LIN {X 0,Y 154.212,Z 695.372,A -85,B 0,C 180,E1 -23468.618,E2 -23468.618} C_VEL
LIN {X 0,Y 158.91,Z 697.062,A -85,B 0,C 180,E1 -23463.751,E2 -23463.751} C_VEL
LIN {X 0,Y 164.977,Z 697.541,A -85,B 0,C 180,E1 -23459.256,E2 -23459.256} C_VEL
LIN {X 0,Y 172.53,Z 696.813,A -85,B 0,C 180,E1 -23455.229,E2 -23455.229} C_VEL
LIN {X 0,Y 181.226,Z 694.851,A -85,B 0,C 180,E1 -23451.648,E2 -23451.648} C_VEL
LIN {X 0,Y 190.909,Z 691.562,A -85,B 0,C 180,E1 -23448.498,E2 -23448.498} C_VEL
LIN {X 0,Y 201.458,Z 686.897,A -85,B 0,C 180,E1 -23445.756,E2 -23445.756} C_VEL
LIN {X 0,Y 207.006,Z 684.055,A -85,B 0,C 180,E1 -23444.523,E2 -23444.523} C_VEL
LIN {X 0,Y 204.306,Z 685.314,A -85,B 0,C 180,E1 -23443.471,E2 -23443.471} C_VEL
LIN {X 0,Y 193.798,Z 689.658,A -85,B 0,C 180,E1 -23440.75,E2 -23440.75} C_VEL
LIN {X 0,Y 188.167,Z 691.451,A -85,B 0,C 180,E1 -23439.054,E2 -23439.054} C_VEL
LIN {X 0,Y 183.778,Z 692.639,A -85,B 0,C 180,E1 -23437.875,E2 -23437.875} C_VEL
LIN {X 0,Y 175.524,Z 694.141,A -85,B 0,C 180,E1 -23436.18,E2 -23436.18} C_VEL
LIN {X 0,Y 169.039,Z 694.749,A -85,B 0,C 180,E1 -23434.699,E2 -23434.699} C_VEL
LIN {X 0,Y 164.24,Z 694.773,A -85,B 0,C 180,E1 -23433.024,E2 -23433.024} C_VEL
LIN {X 0,Y 163.677,Z 694.7,A -85,B 0,C 180,E1 -23432.745,E2 -23432.745} C_VEL
LIN {X 0,Y 157.81,Z 693.959,A -85,B 0,C 180,E1 -23429.333,E2 -23429.333} C_VEL
LIN {X 0,Y 151.671,Z 691.836,A -85,B 0,C 180,E1 -23424.648,E2 -23424.648} C_VEL
LIN {X 0,Y 147.172,Z 688.478,A -85,B 0,C 180,E1 -23419.528,E2 -23419.528} C_VEL
LIN {X 0,Y 144.142,Z 683.771,A -85,B 0,C 180,E1 -23414.11,E2 -23414.11} C_VEL
LIN {X 0,Y 142.894,Z 679.29,A -85,B 0,C 180,E1 -23409.92,E2 -23409.92} C_VEL
LIN {X 0,Y 142.444,Z 672.774,A -85,B 0,C 180,E1 -23404.953,E2 -23404.953} C_VEL
LIN {X 0,Y 142.536,Z 665.887,A -85,B 0,C 180,E1 -23400.706,E2 -23400.706} C_VEL
LIN {X 0,Y 142.741,Z 657.173,A -85,B 0,C 180,E1 -23396.471,E2 -23396.471} C_VEL
LIN {X 0,Y 143.135,Z 648.344,A -85,B 0,C 180,E1 -23392.949,E2 -23392.949} C_VEL
LIN {X 0,Y 143.785,Z 637.536,A -85,B 0,C 180,E1 -23389.412,E2 -23389.412} C_VEL
LIN {X 0,Y 144.647,Z 625.917,A -85,B 0,C 180,E1 -23386.348,E2 -23386.348} C_VEL
LIN {X 0,Y 145.649,Z 612.215,A -85,B 0,C 180,E1 -23383.531,E2 -23383.531} C_VEL
LIN {X 0,Y 146.651,Z 597.973,A -85,B 0,C 180,E1 -23381.307,E2 -23381.307} C_VEL
LIN {X 0,Y 147.514,Z 581.99,A -85,B 0,C 180,E1 -23379.52,E2 -23379.52} C_VEL
LIN {X 0,Y 150.866,Z 512.722,A -85,B 0,C 180,E1 -23373.113,E2 -23373.113} C_VEL
LIN {X 0,Y 150.241,Z 506.777,A -85,B 0,C 180,E1 -23372.506,E2 -23372.506} C_VEL
LIN {X 0,Y 150.609,Z 508.356,A -85,B 0,C 180,E1 -23372.079,E2 -23372.079} C_VEL
LIN {X 0,Y 150.906,Z 508.756,A -85,B 0,C 180,E1 -23371.827,E2 -23371.827} C_VEL
LIN {X 0,Y 151.972,Z 508.48,A -85,B 0,C 180,E1 -23371.11,E2 -23371.11} C_VEL
LIN {X 0,Y 153.68,Z 505.488,A -85,B 0,C 180,E1 -23370.25,E2 -23370.25} C_VEL
LIN {X 0,Y 155.859,Z 499.285,A -85,B 0,C 180,E1 -23369.422,E2 -23369.422} C_VEL
LIN {X 0,Y 157.427,Z 493.941,A -85,B 0,C 180,E1 -23368.928,E2 -23368.928} C_VEL
LIN {X 0,Y 159.201,Z 492.39,A -85,B 0,C 180,E1 -23368.011,E2 -23368.011} C_VEL
LIN {X 0,Y 160.868,Z 489.906,A -85,B 0,C 180,E1 -23367.273,E2 -23367.273} C_VEL
LIN {X 0,Y 163.685,Z 491.039,A -85,B 0,C 180,E1 -23365.68,E2 -23365.68} C_VEL
LIN {X 0,Y 168.067,Z 498.093,A -85,B 0,C 180,E1 -23363.05,E2 -23363.05} C_VEL
LIN {X 0,Y 173.181,Z 507.456,A -85,B 0,C 180,E1 -23360.252,E2 -23360.252} C_VEL
LIN {X 0,Y 177.806,Z 517.181,A -85,B 0,C 180,E1 -23357.91,E2 -23357.91} C_VEL
LIN {X 0,Y 181.79,Z 527.34,A -85,B 0,C 180,E1 -23355.965,E2 -23355.965} C_VEL
LIN {X 0,Y 177.677,Z 588.851,A -85,B 0,C 180,E1 -23353.793,E2 -23353.793} C_VEL
LIN {X 0,Y 175.901,Z 602.055,A -85,B 0,C 180,E1 -23353.016,E2 -23353.016} C_VEL
LIN {X 0,Y 173.476,Z 614.981,A -85,B 0,C 180,E1 -23351.754,E2 -23351.754} C_VEL
LIN {X 0,Y 170.268,Z 627.141,A -85,B 0,C 180,E1 -23350.161,E2 -23350.161} C_VEL
LIN {X 0,Y 166.603,Z 638.578,A -85,B 0,C 180,E1 -23348.094,E2 -23348.094} C_VEL
LIN {X 0,Y 162.567,Z 648.859,A -85,B 0,C 180,E1 -23345.706,E2 -23345.706} C_VEL
LIN {X 0,Y 158.622,Z 658.132,A -85,B 0,C 180,E1 -23342.872,E2 -23342.872} C_VEL
LIN {X 0,Y 154.329,Z 667.038,A -85,B 0,C 180,E1 -23339.311,E2 -23339.311} C_VEL
LIN {X 0,Y 150.538,Z 674.209,A -85,B 0,C 180,E1 -23335.585,E2 -23335.585} C_VEL
LIN {X 0,Y 147.715,Z 679.062,A -85,B 0,C 180,E1 -23332.373,E2 -23332.373} C_VEL
LIN {X 0,Y 145.104,Z 683.747,A -85,B 0,C 180,E1 -23328.35,E2 -23328.35} C_VEL
LIN {X 0,Y 143.11,Z 687.318,A -85,B 0,C 180,E1 -23324.214,E2 -23324.214} C_VEL
LIN {X 0,Y 142.13,Z 689.155,A -85,B 0,C 180,E1 -23321.408,E2 -23321.408} C_VEL
LIN {X 0,Y 141.433,Z 690.53,A -85,B 0,C 180,E1 -23318.573,E2 -23318.573} C_VEL
LIN {X 0,Y 140.948,Z 691.502,A -85,B 0,C 180,E1 -23315.723,E2 -23315.723} C_VEL
LIN {X 0,Y 140.653,Z 692.19,A -85,B 0,C 180,E1 -23312.077,E2 -23312.077} C_VEL
LIN {X 0,Y 140.678,Z 692.063,A -85,B 0,C 180,E1 -23307.136,E2 -23307.136} C_VEL
LIN {X 0,Y 140.948,Z 691.453,A -85,B 0,C 180,E1 -23304.277,E2 -23304.277} C_VEL
LIN {X 0,Y 141.434,Z 690.461,A -85,B 0,C 180,E1 -23301.427,E2 -23301.427} C_VEL
LIN {X 0,Y 142.136,Z 689.046,A -85,B 0,C 180,E1 -23298.593,E2 -23298.593} C_VEL
LIN {X 0,Y 143.725,Z 686.118,A -85,B 0,C 180,E1 -23294.398,E2 -23294.398} C_VEL
LIN {X 0,Y 145.972,Z 682.14,A -85,B 0,C 180,E1 -23290.304,E2 -23290.304} C_VEL
LIN {X 0,Y 148.823,Z 676.997,A -85,B 0,C 180,E1 -23286.334,E2 -23286.334} C_VEL
LIN {X 0,Y 152.409,Z 670.519,A -85,B 0,C 180,E1 -23282.54,E2 -23282.54} C_VEL
LIN {X 0,Y 156.116,Z 663.211,A -85,B 0,C 180,E1 -23279.208,E2 -23279.208} C_VEL
LIN {X 0,Y 160.252,Z 654.194,A -85,B 0,C 180,E1 -23276.002,E2 -23276.002} C_VEL
LIN {X 0,Y 164.398,Z 643.98,A -85,B 0,C 180,E1 -23273.237,E2 -23273.237} C_VEL
LIN {X 0,Y 168.474,Z 632.507,A -85,B 0,C 180,E1 -23270.88,E2 -23270.88} C_VEL
LIN {X 0,Y 171.801,Z 621.001,A -85,B 0,C 180,E1 -23269.116,E2 -23269.116} C_VEL
LIN {X 0,Y 174.716,Z 607.936,A -85,B 0,C 180,E1 -23267.641,E2 -23267.641} C_VEL
LIN {X 0,Y 176.804,Z 595.313,A -85,B 0,C 180,E1 -23266.698,E2 -23266.698} C_VEL
LIN {X 0,Y 178.214,Z 580.651,A -85,B 0,C 180,E1 -23266.047,E2 -23266.047} C_VEL
LIN {X 0,Y 181.605,Z 527.022,A -85,B 0,C 180,E1 -23264.154,E2 -23264.154} C_VEL
LIN {X 0,Y 176.964,Z 515.425,A -85,B 0,C 180,E1 -23261.89,E2 -23261.89} C_VEL
LIN {X 0,Y 171.539,Z 504.437,A -85,B 0,C 180,E1 -23259.109,E2 -23259.109} C_VEL
LIN {X 0,Y 166.539,Z 495.65,A -85,B 0,C 180,E1 -23256.31,E2 -23256.31} C_VEL
LIN {X 0,Y 161.218,Z 487.289,A -85,B 0,C 180,E1 -23252.975,E2 -23252.975} C_VEL
LIN {X 0,Y 157.657,Z 482.205,A -85,B 0,C 180,E1 -23250.469,E2 -23250.469} C_VEL
LIN {X 0,Y 156.455,Z 481.134,A -85,B 0,C 180,E1 -23249.612,E2 -23249.612} C_VEL
LIN {X 0,Y 154.858,Z 481.135,A -85,B 0,C 180,E1 -23248.552,E2 -23248.552} C_VEL
LIN {X 0,Y 151.794,Z 488.731,A -85,B 0,C 180,E1 -23247.125,E2 -23247.125} C_VEL
LIN {X 0,Y 150.556,Z 490.586,A -85,B 0,C 180,E1 -23246.383,E2 -23246.383} C_VEL
LIN {X 0,Y 150.161,Z 490.264,A -85,B 0,C 180,E1 -23246.041,E2 -23246.041} C_VEL
LIN {X 0,Y 149.866,Z 488.044,A -85,B 0,C 180,E1 -23245.567,E2 -23245.567} C_VEL
LIN {X 0,Y 149.888,Z 487.183,A -85,B 0,C 180,E1 -23245.49,E2 -23245.49} C_VEL
LIN {X 0,Y 147.247,Z 543.271,A -85,B 0,C 180,E1 -23240.245,E2 -23240.245} C_VEL
LIN {X 0,Y 146.476,Z 557.446,A -85,B 0,C 180,E1 -23238.534,E2 -23238.534} C_VEL
LIN {X 0,Y 145.519,Z 570.062,A -85,B 0,C 180,E1 -23236.484,E2 -23236.484} C_VEL
LIN {X 0,Y 144.607,Z 581.945,A -85,B 0,C 180,E1 -23234.064,E2 -23234.064} C_VEL
LIN {X 0,Y 143.715,Z 594.089,A -85,B 0,C 180,E1 -23230.952,E2 -23230.952} C_VEL
LIN {X 0,Y 142.872,Z 606.339,A -85,B 0,C 180,E1 -23227.064,E2 -23227.064} C_VEL
LIN {X 0,Y 142.527,Z 617.048,A -85,B 0,C 180,E1 -23222.827,E2 -23222.827} C_VEL
LIN {X 0,Y 142.25,Z 625.752,A -85,B 0,C 180,E1 -23218.585,E2 -23218.585} C_VEL
LIN {X 0,Y 142.882,Z 634.154,A -85,B 0,C 180,E1 -23213.646,E2 -23213.646} C_VEL
LIN {X 0,Y 144.638,Z 641.011,A -85,B 0,C 180,E1 -23208.793,E2 -23208.793} C_VEL
LIN {X 0,Y 147.832,Z 647.241,A -85,B 0,C 180,E1 -23203.427,E2 -23203.427} C_VEL
LIN {X 0,Y 152.456,Z 651.936,A -85,B 0,C 180,E1 -23198.359,E2 -23198.359} C_VEL
LIN {X 0,Y 158.523,Z 655.239,A -85,B 0,C 180,E1 -23193.683,E2 -23193.683} C_VEL
LIN {X 0,Y 165.9,Z 657.207,A -85,B 0,C 180,E1 -23189.446,E2 -23189.446} C_VEL
LIN {X 0,Y 174.366,Z 657.834,A -85,B 0,C 180,E1 -23185.647,E2 -23185.647} C_VEL
LIN {X 0,Y 183.656,Z 657.118,A -85,B 0,C 180,E1 -23182.246,E2 -23182.246} C_VEL
LIN {X 0,Y 193.761,Z 655.054,A -85,B 0,C 180,E1 -23179.24,E2 -23179.24} C_VEL
LIN {X 0,Y 198.138,Z 653.804,A -85,B 0,C 180,E1 -23178.094,E2 -23178.094} C_VEL
LIN {X 0,Y 197.395,Z 654.328,A -85,B 0,C 180,E1 -23177.526,E2 -23177.526} C_VEL
LIN {X 0,Y 187.896,Z 658.559,A -85,B 0,C 180,E1 -23175.29,E2 -23175.29} C_VEL
LIN {X 0,Y 177.607,Z 662.342,A -85,B 0,C 180,E1 -23172.276,E2 -23172.276} C_VEL
LIN {X 0,Y 168.371,Z 664.962,A -85,B 0,C 180,E1 -23168.764,E2 -23168.764} C_VEL
LIN {X 0,Y 160.36,Z 666.488,A -85,B 0,C 180,E1 -23164.733,E2 -23164.733} C_VEL
LIN {X 0,Y 156.579,Z 666.915,A -85,B 0,C 180,E1 -23162.304,E2 -23162.304} C_VEL
LIN {X 0,Y 152.872,Z 673.912,A -85,B 0,C 180,E1 -23159.542,E2 -23159.542} C_VEL
LIN {X 0,Y 149.306,Z 681.107,A -85,B 0,C 180,E1 -23155.811,E2 -23155.811} C_VEL
LIN {X 0,Y 146.611,Z 686.073,A -85,B 0,C 180,E1 -23152.55,E2 -23152.55} C_VEL
LIN {X 0,Y 143.991,Z 690.879,A -85,B 0,C 180,E1 -23148.497,E2 -23148.497} C_VEL
LIN {X 0,Y 142.231,Z 694.562,A -85,B 0,C 180,E1 -23144.304,E2 -23144.304} C_VEL
LIN {X 0,Y 141.421,Z 696.462,A -85,B 0,C 180,E1 -23141.466,E2 -23141.466} C_VEL
LIN {X 0,Y 140.866,Z 697.905,A -85,B 0,C 180,E1 -23138.608,E2 -23138.608} C_VEL
LIN {X 0,Y 140.62,Z 698.923,A -85,B 0,C 180,E1 -23135.737,E2 -23135.737} C_VEL
LIN {X 0,Y 140.587,Z 699.723,A -85,B 0,C 180,E1 -23131.109,E2 -23131.109} C_VEL
LIN {X 0,Y 140.592,Z 699.566,A -85,B 0,C 180,E1 -23127.135,E2 -23127.135} C_VEL
LIN {X 0,Y 140.723,Z 698.951,A -85,B 0,C 180,E1 -23124.267,E2 -23124.267} C_VEL
LIN {X 0,Y 141.103,Z 697.946,A -85,B 0,C 180,E1 -23121.406,E2 -23121.406} C_VEL
LIN {X 0,Y 141.854,Z 696.529,A -85,B 0,C 180,E1 -23118.57,E2 -23118.57} C_VEL
LIN {X 0,Y 143.608,Z 693.574,A -85,B 0,C 180,E1 -23114.385,E2 -23114.385} C_VEL
LIN {X 0,Y 145.115,Z 691.541,A -85,B 0,C 180,E1 -23112.016,E2 -23112.016} C_VEL
LIN {X 0,Y 147.719,Z 694.131,A -85,B 0,C 180,E1 -23107.628,E2 -23107.628} C_VEL
LIN {X 0,Y 152.627,Z 696.23,A -85,B 0,C 180,E1 -23102.582,E2 -23102.582} C_VEL
LIN {X 0,Y 158.935,Z 697.158,A -85,B 0,C 180,E1 -23097.952,E2 -23097.952} C_VEL
LIN {X 0,Y 166.768,Z 696.928,A -85,B 0,C 180,E1 -23093.843,E2 -23093.843} C_VEL
LIN {X 0,Y 175.729,Z 695.482,A -85,B 0,C 180,E1 -23090.216,E2 -23090.216} C_VEL
LIN {X 0,Y 185.696,Z 692.789,A -85,B 0,C 180,E1 -23087.059,E2 -23087.059} C_VEL
LIN {X 0,Y 196.536,Z 688.785,A -85,B 0,C 180,E1 -23084.341,E2 -23084.341} C_VEL
LIN {X 0,Y 193.456,Z 689.867,A -85,B 0,C 180,E1 -23083.4,E2 -23083.4} C_VEL
LIN {X 0,Y 183.305,Z 692.742,A -85,B 0,C 180,E1 -23080.598,E2 -23080.598} C_VEL
LIN {X 0,Y 173.834,Z 694.39,A -85,B 0,C 180,E1 -23077.332,E2 -23077.332} C_VEL
LIN {X 0,Y 165.266,Z 694.806,A -85,B 0,C 180,E1 -23073.561,E2 -23073.561} C_VEL
LIN {X 0,Y 163.677,Z 694.7,A -85,B 0,C 180,E1 -23072.745,E2 -23072.745} C_VEL
LIN {X 0,Y 159.962,Z 694.417,A -85,B 0,C 180,E1 -23071.125,E2 -23071.125} C_VEL
LIN {X 0,Y 152.808,Z 693.264,A -85,B 0,C 180,E1 -23068.653,E2 -23068.653} C_VEL
LIN {X 0,Y 146.216,Z 691.291,A -85,B 0,C 180,E1 -23065.935,E2 -23065.935} C_VEL
LIN {X 0,Y 143.474,Z 689.811,A -85,B 0,C 180,E1 -23063.952,E2 -23063.952} C_VEL
LIN {X 0,Y 139.661,Z 686.102,A -85,B 0,C 180,E1 -23059.092,E2 -23059.092} C_VEL
LIN {X 0,Y 137.477,Z 682.117,A -85,B 0,C 180,E1 -23054.809,E2 -23054.809} C_VEL
LIN {X 0,Y 135.917,Z 675.447,A -85,B 0,C 180,E1 -23048.924,E2 -23048.924} C_VEL
LIN {X 0,Y 135.773,Z 669.278,A -85,B 0,C 180,E1 -23044.453,E2 -23044.453} C_VEL
LIN {X 0,Y 135.872,Z 661.615,A -85,B 0,C 180,E1 -23040,E2 -23040} C_VEL
LIN {X 0,Y 136.019,Z 653.838,A -85,B 0,C 180,E1 -23036.297,E2 -23036.297} C_VEL
LIN {X 0,Y 136.443,Z 644.348,A -85,B 0,C 180,E1 -23032.601,E2 -23032.601} C_VEL
LIN {X 0,Y 137.064,Z 634.008,A -85,B 0,C 180,E1 -23029.288,E2 -23029.288} C_VEL
LIN {X 0,Y 137.99,Z 621.727,A -85,B 0,C 180,E1 -23026.098,E2 -23026.098} C_VEL
LIN {X 0,Y 138.833,Z 608.741,A -85,B 0,C 180,E1 -23023.457,E2 -23023.457} C_VEL
LIN {X 0,Y 139.697,Z 596.213,A -85,B 0,C 180,E1 -23021.483,E2 -23021.483} C_VEL
LIN {X 0,Y 140.791,Z 574.293,A -85,B 0,C 180,E1 -23019.07,E2 -23019.07} C_VEL
LIN {X 0,Y 142.444,Z 537.427,A -85,B 0,C 180,E1 -23015.399,E2 -23015.399} C_VEL
LIN {X 0,Y 142.467,Z 540.512,A -85,B 0,C 180,E1 -23015.014,E2 -23015.014} C_VEL
LIN {X 0,Y 142.752,Z 541.298,A -85,B 0,C 180,E1 -23014.678,E2 -23014.678} C_VEL
LIN {X 0,Y 143.433,Z 541.139,A -85,B 0,C 180,E1 -23014.126,E2 -23014.126} C_VEL
LIN {X 0,Y 144.619,Z 538.864,A -85,B 0,C 180,E1 -23013.418,E2 -23013.418} C_VEL
LIN {X 0,Y 146.697,Z 533.23,A -85,B 0,C 180,E1 -23012.416,E2 -23012.416} C_VEL
LIN {X 0,Y 150.453,Z 520.331,A -85,B 0,C 180,E1 -23011.011,E2 -23011.011} C_VEL
LIN {X 0,Y 151.829,Z 515.486,A -85,B 0,C 180,E1 -23010.54,E2 -23010.54} C_VEL
LIN {X 0,Y 153.658,Z 513.922,A -85,B 0,C 180,E1 -23009.493,E2 -23009.493} C_VEL
LIN {X 0,Y 155.826,Z 510.331,A -85,B 0,C 180,E1 -23008.472,E2 -23008.472} C_VEL
LIN {X 0,Y 158.257,Z 504.284,A -85,B 0,C 180,E1 -23007.562,E2 -23007.562} C_VEL
LIN {X 0,Y 159.969,Z 499.081,A -85,B 0,C 180,E1 -23007.026,E2 -23007.026} C_VEL
LIN {X 0,Y 160.998,Z 497.94,A -85,B 0,C 180,E1 -23006.556,E2 -23006.556} C_VEL
LIN {X 0,Y 161.78,Z 498.314,A -85,B 0,C 180,E1 -23006.109,E2 -23006.109} C_VEL
LIN {X 0,Y 166.905,Z 507.229,A -85,B 0,C 180,E1 -23002.939,E2 -23002.939} C_VEL
LIN {X 0,Y 172.163,Z 517.954,A -85,B 0,C 180,E1 -22999.988,E2 -22999.988} C_VEL
LIN {X 0,Y 176.511,Z 528.678,A -85,B 0,C 180,E1 -22997.691,E2 -22997.691} C_VEL
LIN {X 0,Y 176.81,Z 529.477,A -85,B 0,C 180,E1 -22997.537,E2 -22997.537} C_VEL
LIN {X 0,Y 172.614,Z 589.011,A -85,B 0,C 180,E1 -22995.422,E2 -22995.422} C_VEL
LIN {X 0,Y 170.772,Z 602.284,A -85,B 0,C 180,E1 -22994.631,E2 -22994.631} C_VEL
LIN {X 0,Y 168.257,Z 615.138,A -85,B 0,C 180,E1 -22993.361,E2 -22993.361} C_VEL
LIN {X 0,Y 164.903,Z 627.308,A -85,B 0,C 180,E1 -22991.753,E2 -22991.753} C_VEL
LIN {X 0,Y 161.082,Z 638.752,A -85,B 0,C 180,E1 -22989.65,E2 -22989.65} C_VEL
LIN {X 0,Y 156.865,Z 649.036,A -85,B 0,C 180,E1 -22987.217,E2 -22987.217} C_VEL
LIN {X 0,Y 152.7,Z 658.313,A -85,B 0,C 180,E1 -22984.32,E2 -22984.32} C_VEL
LIN {X 0,Y 148.16,Z 667.222,A -85,B 0,C 180,E1 -22980.659,E2 -22980.659} C_VEL
LIN {X 0,Y 144.171,Z 674.394,A -85,B 0,C 180,E1 -22976.803,E2 -22976.803} C_VEL
LIN {X 0,Y 141.161,Z 679.248,A -85,B 0,C 180,E1 -22973.472,E2 -22973.472} C_VEL
LIN {X 0,Y 138.366,Z 683.935,A -85,B 0,C 180,E1 -22969.278,E2 -22969.278} C_VEL
LIN {X 0,Y 136.218,Z 687.506,A -85,B 0,C 180,E1 -22964.95,E2 -22964.95} C_VEL
LIN {X 0,Y 135.166,Z 689.343,A -85,B 0,C 180,E1 -22962.004,E2 -22962.004} C_VEL
LIN {X 0,Y 134.426,Z 690.718,A -85,B 0,C 180,E1 -22959.024,E2 -22959.024} C_VEL
LIN {X 0,Y 133.603,Z 692.281,A -85,B 0,C 180,E1 -22953.015,E2 -22953.015} C_VEL
LIN {X 0,Y 133.542,Z 692.447,A -85,B 0,C 180,E1 -22949.322,E2 -22949.322} C_VEL
LIN {X 0,Y 133.882,Z 691.642,A -85,B 0,C 180,E1 -22943.974,E2 -22943.974} C_VEL
LIN {X 0,Y 134.427,Z 690.65,A -85,B 0,C 180,E1 -22940.976,E2 -22940.976} C_VEL
LIN {X 0,Y 135.171,Z 689.236,A -85,B 0,C 180,E1 -22937.996,E2 -22937.996} C_VEL
LIN {X 0,Y 136.881,Z 686.308,A -85,B 0,C 180,E1 -22933.597,E2 -22933.597} C_VEL
LIN {X 0,Y 139.3,Z 682.329,A -85,B 0,C 180,E1 -22929.319,E2 -22929.319} C_VEL
LIN {X 0,Y 142.337,Z 677.186,A -85,B 0,C 180,E1 -22925.185,E2 -22925.185} C_VEL
LIN {X 0,Y 146.138,Z 670.707,A -85,B 0,C 180,E1 -22921.255,E2 -22921.255} C_VEL
LIN {X 0,Y 149.799,Z 663.881,A -85,B 0,C 180,E1 -22918.02,E2 -22918.02} C_VEL
LIN {X 0,Y 154.401,Z 654.38,A -85,B 0,C 180,E1 -22914.524,E2 -22914.524} C_VEL
LIN {X 0,Y 158.767,Z 644.164,A -85,B 0,C 180,E1 -22911.704,E2 -22911.704} C_VEL
LIN {X 0,Y 163.031,Z 632.687,A -85,B 0,C 180,E1 -22909.306,E2 -22909.306} C_VEL
LIN {X 0,Y 166.503,Z 621.176,A -85,B 0,C 180,E1 -22907.518,E2 -22907.518} C_VEL
LIN {X 0,Y 169.554,Z 608.102,A -85,B 0,C 180,E1 -22906.029,E2 -22906.029} C_VEL
LIN {X 0,Y 171.754,Z 595.181,A -85,B 0,C 180,E1 -22905.061,E2 -22905.061} C_VEL
LIN {X 0,Y 173.126,Z 581.338,A -85,B 0,C 180,E1 -22904.434,E2 -22904.434} C_VEL
LIN {X 0,Y 176.594,Z 529.191,A -85,B 0,C 180,E1 -22902.576,E2 -22902.576} C_VEL
LIN {X 0,Y 172.028,Z 517.825,A -85,B 0,C 180,E1 -22900.17,E2 -22900.17} C_VEL
LIN {X 0,Y 166.417,Z 506.429,A -85,B 0,C 180,E1 -22897.019,E2 -22897.019} C_VEL
LIN {X 0,Y 161.385,Z 497.781,A -85,B 0,C 180,E1 -22893.899,E2 -22893.899} C_VEL
LIN {X 0,Y 158.043,Z 492.469,A -85,B 0,C 180,E1 -22891.594,E2 -22891.594} C_VEL
LIN {X 0,Y 156.017,Z 489.33,A -85,B 0,C 180,E1 -22890.076,E2 -22890.076} C_VEL
LIN {X 0,Y 155.57,Z 489.422,A -85,B 0,C 180,E1 -22889.798,E2 -22889.798} C_VEL
LIN {X 0,Y 153.336,Z 494.268,A -85,B 0,C 180,E1 -22888.768,E2 -22888.768} C_VEL
LIN {X 0,Y 151.403,Z 496.822,A -85,B 0,C 180,E1 -22887.658,E2 -22887.658} C_VEL
LIN {X 0,Y 150.779,Z 497.545,A -85,B 0,C 180,E1 -22887.274,E2 -22887.274} C_VEL
LIN {X 0,Y 146.646,Z 513.67,A -85,B 0,C 180,E1 -22885.786,E2 -22885.786} C_VEL
LIN {X 0,Y 143.957,Z 522.395,A -85,B 0,C 180,E1 -22884.518,E2 -22884.518} C_VEL
LIN {X 0,Y 142.335,Z 526.521,A -85,B 0,C 180,E1 -22883.556,E2 -22883.556} C_VEL
LIN {X 0,Y 141.607,Z 527.608,A -85,B 0,C 180,E1 -22883.007,E2 -22883.007} C_VEL
LIN {X 0,Y 141.19,Z 527.548,A -85,B 0,C 180,E1 -22882.595,E2 -22882.595} C_VEL
LIN {X 0,Y 140.98,Z 526.456,A -85,B 0,C 180,E1 -22882.244,E2 -22882.244} C_VEL
LIN {X 0,Y 140.994,Z 524.168,A -85,B 0,C 180,E1 -22881.953,E2 -22881.953} C_VEL
LIN {X 0,Y 139.847,Z 549.609,A -85,B 0,C 180,E1 -22879.257,E2 -22879.257} C_VEL
LIN {X 0,Y 139.032,Z 563.216,A -85,B 0,C 180,E1 -22877.276,E2 -22877.276} C_VEL
LIN {X 0,Y 137.983,Z 577.082,A -85,B 0,C 180,E1 -22874.591,E2 -22874.591} C_VEL
LIN {X 0,Y 136.961,Z 589.624,A -85,B 0,C 180,E1 -22871.5,E2 -22871.5} C_VEL
LIN {X 0,Y 136.186,Z 601.705,A -85,B 0,C 180,E1 -22867.786,E2 -22867.786} C_VEL
LIN {X 0,Y 135.732,Z 612.478,A -85,B 0,C 180,E1 -22863.711,E2 -22863.711} C_VEL
LIN {X 0,Y 135.483,Z 620.581,A -85,B 0,C 180,E1 -22860,E2 -22860} C_VEL
LIN {X 0,Y 135.748,Z 629.985,A -85,B 0,C 180,E1 -22854.802,E2 -22854.802} C_VEL
LIN {X 0,Y 137.204,Z 637.739,A -85,B 0,C 180,E1 -22849.672,E2 -22849.672} C_VEL
LIN {X 0,Y 140.136,Z 644.818,A -85,B 0,C 180,E1 -22843.988,E2 -22843.988} C_VEL
LIN {X 0,Y 144.567,Z 650.369,A -85,B 0,C 180,E1 -22838.617,E2 -22838.617} C_VEL
LIN {X 0,Y 148.887,Z 653.572,A -85,B 0,C 180,E1 -22834.86,E2 -22834.86} C_VEL
LIN {X 0,Y 155.887,Z 656.699,A -85,B 0,C 180,E1 -22830.269,E2 -22830.269} C_VEL
LIN {X 0,Y 164.104,Z 658.505,A -85,B 0,C 180,E1 -22826.169,E2 -22826.169} C_VEL
LIN {X 0,Y 173.306,Z 658.97,A -85,B 0,C 180,E1 -22822.534,E2 -22822.534} C_VEL
LIN {X 0,Y 183.318,Z 658.145,A -85,B 0,C 180,E1 -22819.327,E2 -22819.327} C_VEL
LIN {X 0,Y 187.224,Z 657.511,A -85,B 0,C 180,E1 -22818.255,E2 -22818.255} C_VEL
LIN {X 0,Y 186.542,Z 657.918,A -85,B 0,C 180,E1 -22817.722,E2 -22817.722} C_VEL
LIN {X 0,Y 177.579,Z 660.923,A -85,B 0,C 180,E1 -22815.429,E2 -22815.429} C_VEL
LIN {X 0,Y 167.545,Z 663.573,A -85,B 0,C 180,E1 -22812.156,E2 -22812.156} C_VEL
LIN {X 0,Y 158.61,Z 665.153,A -85,B 0,C 180,E1 -22808.341,E2 -22808.341} C_VEL
LIN {X 0,Y 151.228,Z 665.722,A -85,B 0,C 180,E1 -22804.096,E2 -22804.096} C_VEL
LIN {X 0,Y 146.796,Z 673.591,A -85,B 0,C 180,E1 -22800.975,E2 -22800.975} C_VEL
LIN {X 0,Y 142.926,Z 680.918,A -85,B 0,C 180,E1 -22797.055,E2 -22797.055} C_VEL
LIN {X 0,Y 140.03,Z 685.882,A -85,B 0,C 180,E1 -22793.673,E2 -22793.673} C_VEL
LIN {X 0,Y 137.249,Z 690.689,A -85,B 0,C 180,E1 -22789.441,E2 -22789.441} C_VEL
LIN {X 0,Y 135.333,Z 694.372,A -85,B 0,C 180,E1 -22785.05,E2 -22785.05} C_VEL
LIN {X 0,Y 134.452,Z 696.272,A -85,B 0,C 180,E1 -22782.069,E2 -22782.069} C_VEL
LIN {X 0,Y 133.838,Z 697.715,A -85,B 0,C 180,E1 -22779.064,E2 -22779.064} C_VEL
LIN {X 0,Y 133.545,Z 698.734,A -85,B 0,C 180,E1 -22776.042,E2 -22776.042} C_VEL
LIN {X 0,Y 133.542,Z 699.562,A -85,B 0,C 180,E1 -22770.678,E2 -22770.678} C_VEL
LIN {X 0,Y 133.516,Z 699.378,A -85,B 0,C 180,E1 -22766.983,E2 -22766.983} C_VEL
LIN {X 0,Y 134.09,Z 697.757,A -85,B 0,C 180,E1 -22760.953,E2 -22760.953} C_VEL
LIN {X 0,Y 134.889,Z 696.34,A -85,B 0,C 180,E1 -22757.971,E2 -22757.971} C_VEL
LIN {X 0,Y 136.782,Z 693.387,A -85,B 0,C 180,E1 -22753.585,E2 -22753.585} C_VEL
LIN {X 0,Y 139.033,Z 690.433,A -85,B 0,C 180,E1 -22750.242,E2 -22750.242} C_VEL
LIN {X 0,Y 141.33,Z 692.675,A -85,B 0,C 180,E1 -22746.558,E2 -22746.558} C_VEL
LIN {X 0,Y 146.414,Z 695.214,A -85,B 0,C 180,E1 -22741.314,E2 -22741.314} C_VEL
LIN {X 0,Y 152.984,Z 696.583,A -85,B 0,C 180,E1 -22736.545,E2 -22736.545} C_VEL
LIN {X 0,Y 161.111,Z 696.837,A -85,B 0,C 180,E1 -22732.359,E2 -22732.359} C_VEL
LIN {X 0,Y 170.339,Z 695.913,A -85,B 0,C 180,E1 -22728.689,E2 -22728.689} C_VEL
LIN {X 0,Y 180.587,Z 693.78,A -85,B 0,C 180,E1 -22725.531,E2 -22725.531} C_VEL
LIN {X 0,Y 184.301,Z 692.801,A -85,B 0,C 180,E1 -22724.569,E2 -22724.569} C_VEL
LIN {X 0,Y 184.562,Z 692.659,A -85,B 0,C 180,E1 -22723.876,E2 -22723.876} C_VEL
LIN {X 0,Y 178.164,Z 693.928,A -85,B 0,C 180,E1 -22722.113,E2 -22722.113} C_VEL
LIN {X 0,Y 168.263,Z 695.055,A -85,B 0,C 180,E1 -22718.794,E2 -22718.794} C_VEL
LIN {X 0,Y 159.421,Z 694.938,A -85,B 0,C 180,E1 -22714.967,E2 -22714.967} C_VEL
LIN {X 0,Y 151.678,Z 693.613,A -85,B 0,C 180,E1 -22710.643,E2 -22710.643} C_VEL
LIN {X 0,Y 145.303,Z 691.046,A -85,B 0,C 180,E1 -22705.805,E2 -22705.805} C_VEL
LIN {X 0,Y 143.474,Z 689.811,A -85,B 0,C 180,E1 -22703.952,E2 -22703.952} C_VEL
LIN {X 0,Y 141.015,Z 688.176,A -85,B 0,C 180,E1 -22701.897,E2 -22701.897} C_VEL
LIN {X 0,Y 133.941,Z 682.936,A -85,B 0,C 180,E1 -22697.419,E2 -22697.419} C_VEL
LIN {X 0,Y 130.858,Z 679.413,A -85,B 0,C 180,E1 -22694.646,E2 -22694.646} C_VEL
LIN {X 0,Y 130.089,Z 677.629,A -85,B 0,C 180,E1 -22693.13,E2 -22693.13} C_VEL
LIN {X 0,Y 129.138,Z 670.013,A -85,B 0,C 180,E1 -22687.033,E2 -22687.033} C_VEL
LIN {X 0,Y 129.161,Z 664.108,A -85,B 0,C 180,E1 -22683.119,E2 -22683.119} C_VEL
LIN {X 0,Y 129.246,Z 656.887,A -85,B 0,C 180,E1 -22679.221,E2 -22679.221} C_VEL
LIN {X 0,Y 129.474,Z 648.234,A -85,B 0,C 180,E1 -22675.33,E2 -22675.33} C_VEL
LIN {X 0,Y 130.037,Z 636.539,A -85,B 0,C 180,E1 -22671.061,E2 -22671.061} C_VEL
LIN {X 0,Y 130.716,Z 625.962,A -85,B 0,C 180,E1 -22667.975,E2 -22667.975} C_VEL
LIN {X 0,Y 131.496,Z 614.006,A -85,B 0,C 180,E1 -22665.173,E2 -22665.173} C_VEL
LIN {X 0,Y 132.338,Z 601.59,A -85,B 0,C 180,E1 -22662.858,E2 -22662.858} C_VEL
LIN {X 0,Y 133.089,Z 587.635,A -85,B 0,C 180,E1 -22660.929,E2 -22660.929} C_VEL
LIN {X 0,Y 133.823,Z 572.991,A -85,B 0,C 180,E1 -22659.288,E2 -22659.288} C_VEL
LIN {X 0,Y 133.65,Z 576.027,A -85,B 0,C 180,E1 -22659.008,E2 -22659.008} C_VEL
LIN {X 0,Y 133.801,Z 577.477,A -85,B 0,C 180,E1 -22658.629,E2 -22658.629} C_VEL
LIN {X 0,Y 134.263,Z 577.671,A -85,B 0,C 180,E1 -22658.102,E2 -22658.102} C_VEL
LIN {X 0,Y 135.318,Z 575.703,A -85,B 0,C 180,E1 -22657.277,E2 -22657.277} C_VEL
LIN {X 0,Y 137.796,Z 568.432,A -85,B 0,C 180,E1 -22655.819,E2 -22655.819} C_VEL
LIN {X 0,Y 141.164,Z 556.186,A -85,B 0,C 180,E1 -22654.307,E2 -22654.307} C_VEL
LIN {X 0,Y 143.215,Z 548.163,A -85,B 0,C 180,E1 -22653.52,E2 -22653.52} C_VEL
LIN {X 0,Y 144.752,Z 546.737,A -85,B 0,C 180,E1 -22652.471,E2 -22652.471} C_VEL
LIN {X 0,Y 146.703,Z 543.371,A -85,B 0,C 180,E1 -22651.376,E2 -22651.376} C_VEL
LIN {X 0,Y 149.213,Z 536.921,A -85,B 0,C 180,E1 -22650.262,E2 -22650.262} C_VEL
LIN {X 0,Y 152.764,Z 525.481,A -85,B 0,C 180,E1 -22649.014,E2 -22649.014} C_VEL
LIN {X 0,Y 154.101,Z 520.807,A -85,B 0,C 180,E1 -22648.603,E2 -22648.603} C_VEL
LIN {X 0,Y 156.564,Z 517.76,A -85,B 0,C 180,E1 -22647.407,E2 -22647.407} C_VEL
LIN {X 0,Y 159.063,Z 513.27,A -85,B 0,C 180,E1 -22646.38,E2 -22646.38} C_VEL
LIN {X 0,Y 161.18,Z 508.139,A -85,B 0,C 180,E1 -22645.658,E2 -22645.658} C_VEL
LIN {X 0,Y 165.425,Z 516.305,A -85,B 0,C 180,E1 -22642.976,E2 -22642.976} C_VEL
LIN {X 0,Y 169.869,Z 526.241,A -85,B 0,C 180,E1 -22640.378,E2 -22640.378} C_VEL
LIN {X 0,Y 171.942,Z 531.703,A -85,B 0,C 180,E1 -22639.205,E2 -22639.205} C_VEL
LIN {X 0,Y 167.689,Z 589.34,A -85,B 0,C 180,E1 -22637.137,E2 -22637.137} C_VEL
LIN {X 0,Y 165.789,Z 602.519,A -85,B 0,C 180,E1 -22636.343,E2 -22636.343} C_VEL
LIN {X 0,Y 163.175,Z 615.294,A -85,B 0,C 180,E1 -22635.07,E2 -22635.07} C_VEL
LIN {X 0,Y 159.678,Z 627.475,A -85,B 0,C 180,E1 -22633.449,E2 -22633.449} C_VEL
LIN {X 0,Y 155.691,Z 638.925,A -85,B 0,C 180,E1 -22631.314,E2 -22631.314} C_VEL
LIN {X 0,Y 151.273,Z 649.214,A -85,B 0,C 180,E1 -22628.844,E2 -22628.844} C_VEL
LIN {X 0,Y 146.872,Z 658.495,A -85,B 0,C 180,E1 -22625.886,E2 -22625.886} C_VEL
LIN {X 0,Y 142.08,Z 667.406,A -85,B 0,C 180,E1 -22622.124,E2 -22622.124} C_VEL
LIN {X 0,Y 137.87,Z 674.578,A -85,B 0,C 180,E1 -22618.133,E2 -22618.133} C_VEL
LIN {X 0,Y 134.669,Z 679.435,A -85,B 0,C 180,E1 -22614.677,E2 -22614.677} C_VEL
LIN {X 0,Y 131.677,Z 684.122,A -85,B 0,C 180,E1 -22610.299,E2 -22610.299} C_VEL
LIN {X 0,Y 129.361,Z 687.694,A -85,B 0,C 180,E1 -22605.762,E2 -22605.762} C_VEL
LIN {X 0,Y 128.229,Z 689.531,A -85,B 0,C 180,E1 -22602.664,E2 -22602.664} C_VEL
LIN {X 0,Y 127.413,Z 690.907,A -85,B 0,C 180,E1 -22599.525,E2 -22599.525} C_VEL
LIN {X 0,Y 126.515,Z 692.47,A -85,B 0,C 180,E1 -22593.184,E2 -22593.184} C_VEL
LIN {X 0,Y 126.474,Z 692.668,A -85,B 0,C 180,E1 -22590,E2 -22590} C_VEL
LIN {X 0,Y 126.83,Z 691.831,A -85,B 0,C 180,E1 -22583.637,E2 -22583.637} C_VEL
LIN {X 0,Y 127.414,Z 690.839,A -85,B 0,C 180,E1 -22580.475,E2 -22580.475} C_VEL
LIN {X 0,Y 128.234,Z 689.426,A -85,B 0,C 180,E1 -22577.337,E2 -22577.337} C_VEL
LIN {X 0,Y 130.068,Z 686.498,A -85,B 0,C 180,E1 -22572.711,E2 -22572.711} C_VEL
LIN {X 0,Y 132.678,Z 682.519,A -85,B 0,C 180,E1 -22568.235,E2 -22568.235} C_VEL
LIN {X 0,Y 135.92,Z 677.375,A -85,B 0,C 180,E1 -22563.927,E2 -22563.927} C_VEL
LIN {X 0,Y 139.95,Z 670.895,A -85,B 0,C 180,E1 -22559.856,E2 -22559.856} C_VEL
LIN {X 0,Y 144.464,Z 662.864,A -85,B 0,C 180,E1 -22555.997,E2 -22555.997} C_VEL
LIN {X 0,Y 148.665,Z 654.566,A -85,B 0,C 180,E1 -22552.933,E2 -22552.933} C_VEL
LIN {X 0,Y 153.272,Z 644.347,A -85,B 0,C 180,E1 -22550.063,E2 -22550.063} C_VEL
LIN {X 0,Y 157.71,Z 632.867,A -85,B 0,C 180,E1 -22547.622,E2 -22547.622} C_VEL
LIN {X 0,Y 161.339,Z 621.351,A -85,B 0,C 180,E1 -22545.815,E2 -22545.815} C_VEL
LIN {X 0,Y 164.536,Z 608.268,A -85,B 0,C 180,E1 -22544.319,E2 -22544.319} C_VEL
LIN {X 0,Y 166.744,Z 595.834,A -85,B 0,C 180,E1 -22543.37,E2 -22543.37} C_VEL
LIN {X 0,Y 168.275,Z 581.054,A -85,B 0,C 180,E1 -22542.7,E2 -22542.7} C_VEL
LIN {X 0,Y 171.715,Z 531.461,A -85,B 0,C 180,E1 -22540.909,E2 -22540.909} C_VEL
LIN {X 0,Y 167.619,Z 521.198,A -85,B 0,C 180,E1 -22538.572,E2 -22538.572} C_VEL
LIN {X 0,Y 162.716,Z 511.025,A -85,B 0,C 180,E1 -22535.592,E2 -22535.592} C_VEL
LIN {X 0,Y 158.232,Z 503.065,A -85,B 0,C 180,E1 -22532.595,E2 -22532.595} C_VEL
LIN {X 0,Y 155.776,Z 498.924,A -85,B 0,C 180,E1 -22530.783,E2 -22530.783} C_VEL
LIN {X 0,Y 155.462,Z 498.938,A -85,B 0,C 180,E1 -22530.589,E2 -22530.589} C_VEL
LIN {X 0,Y 153.135,Z 502.187,A -85,B 0,C 180,E1 -22529.383,E2 -22529.383} C_VEL
LIN {X 0,Y 148.907,Z 517.733,A -85,B 0,C 180,E1 -22527.954,E2 -22527.954} C_VEL
LIN {X 0,Y 146.031,Z 526.443,A -85,B 0,C 180,E1 -22526.692,E2 -22526.692} C_VEL
LIN {X 0,Y 143.992,Z 531.235,A -85,B 0,C 180,E1 -22525.572,E2 -22525.572} C_VEL
LIN {X 0,Y 142.324,Z 533.759,A -85,B 0,C 180,E1 -22524.429,E2 -22524.429} C_VEL
LIN {X 0,Y 141.505,Z 534.678,A -85,B 0,C 180,E1 -22523.8,E2 -22523.8} C_VEL
LIN {X 0,Y 138.142,Z 548.506,A -85,B 0,C 180,E1 -22522.332,E2 -22522.332} C_VEL
LIN {X 0,Y 135.547,Z 557.291,A -85,B 0,C 180,E1 -22520.806,E2 -22520.806} C_VEL
LIN {X 0,Y 133.646,Z 562.49,A -85,B 0,C 180,E1 -22519.378,E2 -22519.378} C_VEL
LIN {X 0,Y 132.521,Z 564.816,A -85,B 0,C 180,E1 -22518.334,E2 -22518.334} C_VEL
LIN {X 0,Y 132.035,Z 565.154,A -85,B 0,C 180,E1 -22517.742,E2 -22517.742} C_VEL
LIN {X 0,Y 131.889,Z 564.238,A -85,B 0,C 180,E1 -22517.377,E2 -22517.377} C_VEL
LIN {X 0,Y 132.139,Z 561.209,A -85,B 0,C 180,E1 -22517.124,E2 -22517.124} C_VEL
LIN {X 0,Y 131.078,Z 575.331,A -85,B 0,C 180,E1 -22514.353,E2 -22514.353} C_VEL
LIN {X 0,Y 130.02,Z 588.929,A -85,B 0,C 180,E1 -22510.905,E2 -22510.905} C_VEL
LIN {X 0,Y 129.269,Z 601.029,A -85,B 0,C 180,E1 -22507.027,E2 -22507.027} C_VEL
LIN {X 0,Y 128.933,Z 611.078,A -85,B 0,C 180,E1 -22503.125,E2 -22503.125} C_VEL
LIN {X 0,Y 128.693,Z 619.37,A -85,B 0,C 180,E1 -22499.218,E2 -22499.218} C_VEL
LIN {X 0,Y 129.059,Z 629.053,A -85,B 0,C 180,E1 -22493.748,E2 -22493.748} C_VEL
LIN {X 0,Y 130.7,Z 637.035,A -85,B 0,C 180,E1 -22488.367,E2 -22488.367} C_VEL
LIN {X 0,Y 133.431,Z 643.589,A -85,B 0,C 180,E1 -22483.161,E2 -22483.161} C_VEL
LIN {X 0,Y 138.012,Z 649.62,A -85,B 0,C 180,E1 -22477.547,E2 -22477.547} C_VEL
LIN {X 0,Y 142.51,Z 653.179,A -85,B 0,C 180,E1 -22473.651,E2 -22473.651} C_VEL
LIN {X 0,Y 149.757,Z 656.801,A -85,B 0,C 180,E1 -22468.921,E2 -22468.921} C_VEL
LIN {X 0,Y 158.264,Z 659.096,A -85,B 0,C 180,E1 -22464.74,E2 -22464.74} C_VEL
LIN {X 0,Y 167.779,Z 660.095,A -85,B 0,C 180,E1 -22461.073,E2 -22461.073} C_VEL
LIN {X 0,Y 175.758,Z 660.017,A -85,B 0,C 180,E1 -22458.55,E2 -22458.55} C_VEL
LIN {X 0,Y 174.661,Z 660.542,A -85,B 0,C 180,E1 -22457.631,E2 -22457.631} C_VEL
LIN {X 0,Y 167.388,Z 662.213,A -85,B 0,C 180,E1 -22455.543,E2 -22455.543} C_VEL
LIN {X 0,Y 157.609,Z 663.819,A -85,B 0,C 180,E1 -22451.98,E2 -22451.98} C_VEL
LIN {X 0,Y 149.016,Z 664.423,A -85,B 0,C 180,E1 -22447.815,E2 -22447.815} C_VEL
LIN {X 0,Y 146.053,Z 664.507,A -85,B 0,C 180,E1 -22446.012,E2 -22446.012} C_VEL
LIN {X 0,Y 141.555,Z 672.047,A -85,B 0,C 180,E1 -22443.102,E2 -22443.102} C_VEL
LIN {X 0,Y 137.639,Z 678.888,A -85,B 0,C 180,E1 -22439.568,E2 -22439.568} C_VEL
LIN {X 0,Y 134.673,Z 683.828,A -85,B 0,C 180,E1 -22436.332,E2 -22436.332} C_VEL
LIN {X 0,Y 131.476,Z 689.049,A -85,B 0,C 180,E1 -22431.974,E2 -22431.974} C_VEL
LIN {X 0,Y 129.037,Z 693.093,A -85,B 0,C 180,E1 -22427.431,E2 -22427.431} C_VEL
LIN {X 0,Y 127.479,Z 696.082,A -85,B 0,C 180,E1 -22422.74,E2 -22422.74} C_VEL
LIN {X 0,Y 126.805,Z 697.525,A -85,B 0,C 180,E1 -22419.571,E2 -22419.571} C_VEL
LIN {X 0,Y 126.465,Z 698.544,A -85,B 0,C 180,E1 -22416.381,E2 -22416.381} C_VEL
LIN {X 0,Y 126.378,Z 699.172,A -85,B 0,C 180,E1 -22413.188,E2 -22413.188} C_VEL
LIN {X 0,Y 126.504,Z 699.406,A -85,B 0,C 180,E1 -22410,E2 -22410} C_VEL
LIN {X 0,Y 126.444,Z 699.189,A -85,B 0,C 180,E1 -22406.814,E2 -22406.814} C_VEL
LIN {X 0,Y 127.076,Z 697.569,A -85,B 0,C 180,E1 -22400.449,E2 -22400.449} C_VEL
LIN {X 0,Y 127.951,Z 696.152,A -85,B 0,C 180,E1 -22397.308,E2 -22397.308} C_VEL
LIN {X 0,Y 129.992,Z 693.2,A -85,B 0,C 180,E1 -22392.701,E2 -22392.701} C_VEL
LIN {X 0,Y 133.189,Z 689.225,A -85,B 0,C 180,E1 -22388.221,E2 -22388.221} C_VEL
LIN {X 0,Y 137.494,Z 692.673,A -85,B 0,C 180,E1 -22382.61,E2 -22382.61} C_VEL
LIN {X 0,Y 143.506,Z 695.024,A -85,B 0,C 180,E1 -22377.404,E2 -22377.404} C_VEL
LIN {X 0,Y 151.207,Z 696.297,A -85,B 0,C 180,E1 -22372.826,E2 -22372.826} C_VEL
LIN {X 0,Y 160.2,Z 696.462,A -85,B 0,C 180,E1 -22368.848,E2 -22368.848} C_VEL
LIN {X 0,Y 170.225,Z 695.479,A -85,B 0,C 180,E1 -22365.423,E2 -22365.423} C_VEL
LIN {X 0,Y 173.458,Z 694.963,A -85,B 0,C 180,E1 -22364.504,E2 -22364.504} C_VEL
LIN {X 0,Y 173.004,Z 694.933,A -85,B 0,C 180,E1 -22363.677,E2 -22363.677} C_VEL
LIN {X 0,Y 162.811,Z 695.497,A -85,B 0,C 180,E1 -22360.353,E2 -22360.353} C_VEL
LIN {X 0,Y 153.667,Z 694.864,A -85,B 0,C 180,E1 -22356.481,E2 -22356.481} C_VEL
LIN {X 0,Y 145.653,Z 693.04,A -85,B 0,C 180,E1 -22352.057,E2 -22352.057} C_VEL
LIN {X 0,Y 139.035,Z 690.034,A -85,B 0,C 180,E1 -22347.061,E2 -22347.061} C_VEL
LIN {X 0,Y 134.117,Z 685.815,A -85,B 0,C 180,E1 -22341.519,E2 -22341.519} C_VEL
LIN {X 0,Y 130.886,Z 680.227,A -85,B 0,C 180,E1 -22335.574,E2 -22335.574} C_VEL
LIN {X 0,Y 130.089,Z 677.629,A -85,B 0,C 180,E1 -22333.13,E2 -22333.13} C_VEL
LIN {X 0,Y 128.984,Z 674.776,A -85,B 0,C 180,E1 -22330.905,E2 -22330.905} C_VEL
LIN {X 0,Y 125.956,Z 669.1,A -85,B 0,C 180,E1 -22327.514,E2 -22327.514} C_VEL
LIN {X 0,Y 123.633,Z 664.045,A -85,B 0,C 180,E1 -22324.845,E2 -22324.845} C_VEL
LIN {X 0,Y 122.693,Z 660.141,A -85,B 0,C 180,E1 -22322.769,E2 -22322.769} C_VEL
LIN {X 0,Y 122.634,Z 658.846,A -85,B 0,C 180,E1 -22322.058,E2 -22322.058} C_VEL
LIN {X 0,Y 122.668,Z 651.631,A -85,B 0,C 180,E1 -22318.358,E2 -22318.358} C_VEL
LIN {X 0,Y 122.965,Z 641.879,A -85,B 0,C 180,E1 -22314.259,E2 -22314.259} C_VEL
LIN {X 0,Y 123.466,Z 631.253,A -85,B 0,C 180,E1 -22310.581,E2 -22310.581} C_VEL
LIN {X 0,Y 124.224,Z 619.721,A -85,B 0,C 180,E1 -22307.336,E2 -22307.336} C_VEL
LIN {X 0,Y 124.965,Z 606.952,A -85,B 0,C 180,E1 -22304.511,E2 -22304.511} C_VEL
LIN {X 0,Y 125.243,Z 603.053,A -85,B 0,C 180,E1 -22303.705,E2 -22303.705} C_VEL
LIN {X 0,Y 125.041,Z 604.85,A -85,B 0,C 180,E1 -22303.216,E2 -22303.216} C_VEL
LIN {X 0,Y 125.186,Z 605.308,A -85,B 0,C 180,E1 -22302.773,E2 -22302.773} C_VEL
LIN {X 0,Y 126.015,Z 604.847,A -85,B 0,C 180,E1 -22301.778,E2 -22301.778} C_VEL
LIN {X 0,Y 127.541,Z 602.607,A -85,B 0,C 180,E1 -22300.589,E2 -22300.589} C_VEL
LIN {X 0,Y 129.984,Z 597.52,A -85,B 0,C 180,E1 -22299.217,E2 -22299.217} C_VEL
LIN {X 0,Y 132.442,Z 590.41,A -85,B 0,C 180,E1 -22298.092,E2 -22298.092} C_VEL
LIN {X 0,Y 133.965,Z 584.643,A -85,B 0,C 180,E1 -22297.441,E2 -22297.441} C_VEL
LIN {X 0,Y 135.536,Z 582.999,A -85,B 0,C 180,E1 -22296.102,E2 -22296.102} C_VEL
LIN {X 0,Y 137.316,Z 579.55,A -85,B 0,C 180,E1 -22294.888,E2 -22294.888} C_VEL
LIN {X 0,Y 140.222,Z 571.399,A -85,B 0,C 180,E1 -22293.359,E2 -22293.359} C_VEL
LIN {X 0,Y 143.73,Z 559.289,A -85,B 0,C 180,E1 -22291.925,E2 -22291.925} C_VEL
LIN {X 0,Y 145.307,Z 553.387,A -85,B 0,C 180,E1 -22291.371,E2 -22291.371} C_VEL
LIN {X 0,Y 147.835,Z 549.849,A -85,B 0,C 180,E1 -22289.957,E2 -22289.957} C_VEL
LIN {X 0,Y 150.045,Z 545.36,A -85,B 0,C 180,E1 -22288.931,E2 -22288.931} C_VEL
LIN {X 0,Y 153.022,Z 537.514,A -85,B 0,C 180,E1 -22287.797,E2 -22287.797} C_VEL
LIN {X 0,Y 156.918,Z 525.276,A -85,B 0,C 180,E1 -22286.586,E2 -22286.586} C_VEL
LIN {X 0,Y 160.319,Z 520.362,A -85,B 0,C 180,E1 -22285.159,E2 -22285.159} C_VEL
LIN {X 0,Y 161.063,Z 519.391,A -85,B 0,C 180,E1 -22284.853,E2 -22284.853} C_VEL
LIN {X 0,Y 165.698,Z 529.964,A -85,B 0,C 180,E1 -22281.898,E2 -22281.898} C_VEL
LIN {X 0,Y 167.16,Z 533.953,A -85,B 0,C 180,E1 -22280.994,E2 -22280.994} C_VEL
LIN {X 0,Y 165.772,Z 553.605,A -85,B 0,C 180,E1 -22280.265,E2 -22280.265} C_VEL
LIN {X 0,Y 162.8,Z 590.656,A -85,B 0,C 180,E1 -22278.918,E2 -22278.918} C_VEL
LIN {X 0,Y 160.765,Z 603.717,A -85,B 0,C 180,E1 -22278.081,E2 -22278.081} C_VEL
LIN {X 0,Y 157.987,Z 616.534,A -85,B 0,C 180,E1 -22276.756,E2 -22276.756} C_VEL
LIN {X 0,Y 154.619,Z 627.641,A -85,B 0,C 180,E1 -22275.252,E2 -22275.252} C_VEL
LIN {X 0,Y 150.442,Z 639.099,A -85,B 0,C 180,E1 -22273.096,E2 -22273.096} C_VEL
LIN {X 0,Y 145.83,Z 649.391,A -85,B 0,C 180,E1 -22270.588,E2 -22270.588} C_VEL
LIN {X 0,Y 141.172,Z 658.676,A -85,B 0,C 180,E1 -22267.579,E2 -22267.579} C_VEL
LIN {X 0,Y 136.106,Z 667.59,A -85,B 0,C 180,E1 -22263.717,E2 -22263.717} C_VEL
LIN {X 0,Y 131.639,Z 674.764,A -85,B 0,C 180,E1 -22259.594,E2 -22259.594} C_VEL
LIN {X 0,Y 128.247,Z 679.62,A -85,B 0,C 180,E1 -22256.002,E2 -22256.002} C_VEL
LIN {X 0,Y 125.038,Z 684.309,A -85,B 0,C 180,E1 -22251.429,E2 -22251.429} C_VEL
LIN {X 0,Y 122.54,Z 687.882,A -85,B 0,C 180,E1 -22246.664,E2 -22246.664} C_VEL
LIN {X 0,Y 121.322,Z 689.719,A -85,B 0,C 180,E1 -22243.398,E2 -22243.398} C_VEL
LIN {X 0,Y 120.428,Z 691.095,A -85,B 0,C 180,E1 -22240.083,E2 -22240.083} C_VEL
LIN {X 0,Y 119.44,Z 692.658,A -85,B 0,C 180,E1 -22233.373,E2 -22233.373} C_VEL
LIN {X 0,Y 119.394,Z 692.857,A -85,B 0,C 180,E1 -22230,E2 -22230} C_VEL
LIN {X 0,Y 119.44,Z 692.63,A -85,B 0,C 180,E1 -22226.627,E2 -22226.627} C_VEL
LIN {X 0,Y 120.429,Z 691.028,A -85,B 0,C 180,E1 -22219.917,E2 -22219.917} C_VEL
LIN {X 0,Y 121.327,Z 689.615,A -85,B 0,C 180,E1 -22216.602,E2 -22216.602} C_VEL
LIN {X 0,Y 123.291,Z 686.688,A -85,B 0,C 180,E1 -22211.728,E2 -22211.728} C_VEL
LIN {X 0,Y 126.089,Z 682.709,A -85,B 0,C 180,E1 -22207.035,E2 -22207.035} C_VEL
LIN {X 0,Y 129.579,Z 677.563,A -85,B 0,C 180,E1 -22202.547,E2 -22202.547} C_VEL
LIN {X 0,Y 133.853,Z 671.084,A -85,B 0,C 180,E1 -22198.328,E2 -22198.328} C_VEL
LIN {X 0,Y 138.362,Z 663.524,A -85,B 0,C 180,E1 -22194.565,E2 -22194.565} C_VEL
LIN {X 0,Y 143.074,Z 654.751,A -85,B 0,C 180,E1 -22191.222,E2 -22191.222} C_VEL
LIN {X 0,Y 147.915,Z 644.53,A -85,B 0,C 180,E1 -22188.303,E2 -22188.303} C_VEL
LIN {X 0,Y 152.546,Z 633.047,A -85,B 0,C 180,E1 -22185.826,E2 -22185.826} C_VEL
LIN {X 0,Y 156.326,Z 621.526,A -85,B 0,C 180,E1 -22184.002,E2 -22184.002} C_VEL
LIN {X 0,Y 159.67,Z 608.434,A -85,B 0,C 180,E1 -22182.501,E2 -22182.501} C_VEL
LIN {X 0,Y 161.976,Z 595.86,A -85,B 0,C 180,E1 -22181.541,E2 -22181.541} C_VEL
LIN {X 0,Y 163.55,Z 581.12,A -85,B 0,C 180,E1 -22180.871,E2 -22180.871} C_VEL
LIN {X 0,Y 166.988,Z 533.745,A -85,B 0,C 180,E1 -22179.147,E2 -22179.147} C_VEL
LIN {X 0,Y 163.505,Z 525.052,A -85,B 0,C 180,E1 -22176.997,E2 -22176.997} C_VEL
LIN {X 0,Y 159.475,Z 516.306,A -85,B 0,C 180,E1 -22174.342,E2 -22174.342} C_VEL
LIN {X 0,Y 155.324,Z 508.583,A -85,B 0,C 180,E1 -22171.356,E2 -22171.356} C_VEL
LIN {X 0,Y 155.227,Z 508.446,A -85,B 0,C 180,E1 -22171.285,E2 -22171.285} C_VEL
LIN {X 0,Y 151.19,Z 522.322,A -85,B 0,C 180,E1 -22169.981,E2 -22169.981} C_VEL
LIN {X 0,Y 148.119,Z 530.947,A -85,B 0,C 180,E1 -22168.713,E2 -22168.713} C_VEL
LIN {X 0,Y 145.83,Z 535.965,A -85,B 0,C 180,E1 -22167.548,E2 -22167.548} C_VEL
LIN {X 0,Y 143.44,Z 539.673,A -85,B 0,C 180,E1 -22166.068,E2 -22166.068} C_VEL
LIN {X 0,Y 140.178,Z 552.135,A -85,B 0,C 180,E1 -22164.729,E2 -22164.729} C_VEL
LIN {X 0,Y 137.366,Z 561.032,A -85,B 0,C 180,E1 -22163.222,E2 -22163.222} C_VEL
LIN {X 0,Y 135.059,Z 566.929,A -85,B 0,C 180,E1 -22161.663,E2 -22161.663} C_VEL
LIN {X 0,Y 133.424,Z 570.21,A -85,B 0,C 180,E1 -22160.317,E2 -22160.317} C_VEL
LIN {X 0,Y 132.04,Z 571.947,A -85,B 0,C 180,E1 -22158.907,E2 -22158.907} C_VEL
LIN {X 0,Y 131.574,Z 572.47,A -85,B 0,C 180,E1 -22158.39,E2 -22158.39} C_VEL
LIN {X 0,Y 128.506,Z 583.026,A -85,B 0,C 180,E1 -22155.934,E2 -22155.934} C_VEL
LIN {X 0,Y 125.968,Z 590.703,A -85,B 0,C 180,E1 -22153.45,E2 -22153.45} C_VEL
LIN {X 0,Y 123.811,Z 596.026,A -85,B 0,C 180,E1 -22150.942,E2 -22150.942} C_VEL
LIN {X 0,Y 122.753,Z 598.071,A -85,B 0,C 180,E1 -22149.267,E2 -22149.267} C_VEL
LIN {X 0,Y 122.345,Z 598.478,A -85,B 0,C 180,E1 -22148.257,E2 -22148.257} C_VEL
LIN {X 0,Y 122.324,Z 597.998,A -85,B 0,C 180,E1 -22147.843,E2 -22147.843} C_VEL
LIN {X 0,Y 122.62,Z 596.514,A -85,B 0,C 180,E1 -22147.513,E2 -22147.513} C_VEL
LIN {X 0,Y 122.157,Z 607.501,A -85,B 0,C 180,E1 -22143.298,E2 -22143.298} C_VEL
LIN {X 0,Y 122.036,Z 614.763,A -85,B 0,C 180,E1 -22140,E2 -22140} C_VEL
LIN {X 0,Y 122.191,Z 625.335,A -85,B 0,C 180,E1 -22134.223,E2 -22134.223} C_VEL
LIN {X 0,Y 123.642,Z 634.014,A -85,B 0,C 180,E1 -22128.525,E2 -22128.525} C_VEL
LIN {X 0,Y 126.8,Z 642.131,A -85,B 0,C 180,E1 -22122.251,E2 -22122.251} C_VEL
LIN {X 0,Y 131.55,Z 648.623,A -85,B 0,C 180,E1 -22116.379,E2 -22116.379} C_VEL
LIN {X 0,Y 137.955,Z 653.694,A -85,B 0,C 180,E1 -22111.055,E2 -22111.055} C_VEL
LIN {X 0,Y 143.717,Z 656.662,A -85,B 0,C 180,E1 -22107.458,E2 -22107.458} C_VEL
LIN {X 0,Y 152.533,Z 659.459,A -85,B 0,C 180,E1 -22103.203,E2 -22103.203} C_VEL
LIN {X 0,Y 162.351,Z 660.998,A -85,B 0,C 180,E1 -22099.508,E2 -22099.508} C_VEL
LIN {X 0,Y 164.999,Z 661.215,A -85,B 0,C 180,E1 -22098.651,E2 -22098.651} C_VEL
LIN {X 0,Y 164.124,Z 661.573,A -85,B 0,C 180,E1 -22097.809,E2 -22097.809} C_VEL
LIN {X 0,Y 152.449,Z 662.926,A -85,B 0,C 180,E1 -22093.75,E2 -22093.75} C_VEL
LIN {X 0,Y 143.58,Z 663.094,A -85,B 0,C 180,E1 -22089.519,E2 -22089.519} C_VEL
LIN {X 0,Y 141.213,Z 663.003,A -85,B 0,C 180,E1 -22088.13,E2 -22088.13} C_VEL
LIN {X 0,Y 136.559,Z 670.392,A -85,B 0,C 180,E1 -22085.379,E2 -22085.379} C_VEL
LIN {X 0,Y 131.934,Z 677.961,A -85,B 0,C 180,E1 -22081.537,E2 -22081.537} C_VEL
LIN {X 0,Y 128.343,Z 683.639,A -85,B 0,C 180,E1 -22077.74,E2 -22077.74} C_VEL
LIN {X 0,Y 124.9,Z 688.859,A -85,B 0,C 180,E1 -22073.196,E2 -22073.196} C_VEL
LIN {X 0,Y 122.232,Z 692.903,A -85,B 0,C 180,E1 -22068.435,E2 -22068.435} C_VEL
LIN {X 0,Y 120.535,Z 695.891,A -85,B 0,C 180,E1 -22063.487,E2 -22063.487} C_VEL
LIN {X 0,Y 119.796,Z 697.335,A -85,B 0,C 180,E1 -22060.137,E2 -22060.137} C_VEL
LIN {X 0,Y 119.411,Z 698.354,A -85,B 0,C 180,E1 -22056.76,E2 -22056.76} C_VEL
LIN {X 0,Y 119.285,Z 698.982,A -85,B 0,C 180,E1 -22053.378,E2 -22053.378} C_VEL
LIN {X 0,Y 119.4,Z 699.217,A -85,B 0,C 180,E1 -22050,E2 -22050} C_VEL
LIN {X 0,Y 119.36,Z 699,A -85,B 0,C 180,E1 -22046.624,E2 -22046.624} C_VEL
LIN {X 0,Y 120.068,Z 697.38,A -85,B 0,C 180,E1 -22039.886,E2 -22039.886} C_VEL
LIN {X 0,Y 121.041,Z 695.964,A -85,B 0,C 180,E1 -22036.57,E2 -22036.57} C_VEL
LIN {X 0,Y 123.24,Z 693.012,A -85,B 0,C 180,E1 -22031.721,E2 -22031.721} C_VEL
LIN {X 0,Y 127.342,Z 688.017,A -85,B 0,C 180,E1 -22026.198,E2 -22026.198} C_VEL
LIN {X 0,Y 134.347,Z 692.555,A -85,B 0,C 180,E1 -22018.458,E2 -22018.458} C_VEL
LIN {X 0,Y 141.469,Z 694.778,A -85,B 0,C 180,E1 -22013.405,E2 -22013.405} C_VEL
LIN {X 0,Y 150.163,Z 695.976,A -85,B 0,C 180,E1 -22009.062,E2 -22009.062} C_VEL
LIN {X 0,Y 159.964,Z 696.084,A -85,B 0,C 180,E1 -22005.335,E2 -22005.335} C_VEL
LIN {X 0,Y 162.605,Z 695.848,A -85,B 0,C 180,E1 -22003.752,E2 -22003.752} C_VEL
LIN {X 0,Y 152.621,Z 695.276,A -85,B 0,C 180,E1 -22000.142,E2 -22000.142} C_VEL
LIN {X 0,Y 143.73,Z 693.555,A -85,B 0,C 180,E1 -21995.928,E2 -21995.928} C_VEL
LIN {X 0,Y 136.058,Z 690.658,A -85,B 0,C 180,E1 -21991.101,E2 -21991.101} C_VEL
LIN {X 0,Y 130.104,Z 686.629,A -85,B 0,C 180,E1 -21985.604,E2 -21985.604} C_VEL
LIN {X 0,Y 125.782,Z 681.313,A -85,B 0,C 180,E1 -21979.587,E2 -21979.587} C_VEL
LIN {X 0,Y 123.402,Z 674.574,A -85,B 0,C 180,E1 -21973.168,E2 -21973.168} C_VEL
LIN {X 0,Y 122.61,Z 667.279,A -85,B 0,C 180,E1 -21967.41,E2 -21967.41} C_VEL
LIN {X 0,Y 122.627,Z 659.576,A -85,B 0,C 180,E1 -21962.463,E2 -21962.463} C_VEL
LIN {X 0,Y 122.634,Z 658.846,A -85,B 0,C 180,E1 -21962.058,E2 -21962.058} C_VEL
LIN {X 0,Y 122.045,Z 654.84,A -85,B 0,C 180,E1 -21960.085,E2 -21960.085} C_VEL
LIN {X 0,Y 120.588,Z 650.403,A -85,B 0,C 180,E1 -21958.34,E2 -21958.34} C_VEL
LIN {X 0,Y 116.883,Z 639.239,A -85,B 0,C 180,E1 -21954.594,E2 -21954.594} C_VEL
LIN {X 0,Y 116.549,Z 634.295,A -85,B 0,C 180,E1 -21952.916,E2 -21952.916} C_VEL
LIN {X 0,Y 117.207,Z 622.513,A -85,B 0,C 180,E1 -21949.2,E2 -21949.2} C_VEL
LIN {X 0,Y 117.403,Z 618.94,A -85,B 0,C 180,E1 -21948.234,E2 -21948.234} C_VEL
LIN {X 0,Y 117.171,Z 619.693,A -85,B 0,C 180,E1 -21947.881,E2 -21947.881} C_VEL
LIN {X 0,Y 117.613,Z 620.445,A -85,B 0,C 180,E1 -21946.171,E2 -21946.171} C_VEL
LIN {X 0,Y 119.11,Z 618.856,A -85,B 0,C 180,E1 -21944.602,E2 -21944.602} C_VEL
LIN {X 0,Y 121.863,Z 614.822,A -85,B 0,C 180,E1 -21942.808,E2 -21942.808} C_VEL
LIN {X 0,Y 123.594,Z 612.026,A -85,B 0,C 180,E1 -21941.775,E2 -21941.775} C_VEL
LIN {X 0,Y 125.035,Z 611.056,A -85,B 0,C 180,E1 -21940.29,E2 -21940.29} C_VEL
LIN {X 0,Y 126.915,Z 608.96,A -85,B 0,C 180,E1 -21938.903,E2 -21938.903} C_VEL
LIN {X 0,Y 129.516,Z 604.868,A -85,B 0,C 180,E1 -21937.465,E2 -21937.465} C_VEL
LIN {X 0,Y 132.598,Z 598.488,A -85,B 0,C 180,E1 -21936.162,E2 -21936.162} C_VEL
LIN {X 0,Y 135.664,Z 589.801,A -85,B 0,C 180,E1 -21935.005,E2 -21935.005} C_VEL
LIN {X 0,Y 138.035,Z 586.414,A -85,B 0,C 180,E1 -21933.442,E2 -21933.442} C_VEL
LIN {X 0,Y 140.29,Z 581.507,A -85,B 0,C 180,E1 -21932.192,E2 -21932.192} C_VEL
LIN {X 0,Y 143.599,Z 572.226,A -85,B 0,C 180,E1 -21930.697,E2 -21930.697} C_VEL
LIN {X 0,Y 147.86,Z 557.771,A -85,B 0,C 180,E1 -21929.193,E2 -21929.193} C_VEL
LIN {X 0,Y 150.797,Z 553.279,A -85,B 0,C 180,E1 -21927.758,E2 -21927.758} C_VEL
LIN {X 0,Y 154.124,Z 546.143,A -85,B 0,C 180,E1 -21926.429,E2 -21926.429} C_VEL
LIN {X 0,Y 157.776,Z 535.949,A -85,B 0,C 180,E1 -21925.269,E2 -21925.269} C_VEL
LIN {X 0,Y 159.773,Z 529.653,A -85,B 0,C 180,E1 -21924.725,E2 -21924.725} C_VEL
LIN {X 0,Y 160.384,Z 530.543,A -85,B 0,C 180,E1 -21924.35,E2 -21924.35} C_VEL
LIN {X 0,Y 162.695,Z 536.656,A -85,B 0,C 180,E1 -21922.788,E2 -21922.788} C_VEL
LIN {X 0,Y 158.275,Z 590.36,A -85,B 0,C 180,E1 -21920.871,E2 -21920.871} C_VEL
LIN {X 0,Y 156.216,Z 603.439,A -85,B 0,C 180,E1 -21920.047,E2 -21920.047} C_VEL
LIN {X 0,Y 153.225,Z 616.692,A -85,B 0,C 180,E1 -21918.684,E2 -21918.684} C_VEL
LIN {X 0,Y 149.716,Z 627.808,A -85,B 0,C 180,E1 -21917.178,E2 -21917.178} C_VEL
LIN {X 0,Y 145.349,Z 639.273,A -85,B 0,C 180,E1 -21915.004,E2 -21915.004} C_VEL
LIN {X 0,Y 140.514,Z 649.569,A -85,B 0,C 180,E1 -21912.472,E2 -21912.472} C_VEL
LIN {X 0,Y 135.602,Z 658.857,A -85,B 0,C 180,E1 -21909.412,E2 -21909.412} C_VEL
LIN {X 0,Y 130.254,Z 667.773,A -85,B 0,C 180,E1 -21905.453,E2 -21905.453} C_VEL
LIN {X 0,Y 125.499,Z 674.949,A -85,B 0,C 180,E1 -21901.199,E2 -21901.199} C_VEL
LIN {X 0,Y 121.907,Z 679.806,A -85,B 0,C 180,E1 -21897.465,E2 -21897.465} C_VEL
LIN {X 0,Y 118.454,Z 684.496,A -85,B 0,C 180,E1 -21892.684,E2 -21892.684} C_VEL
LIN {X 0,Y 115.76,Z 688.069,A -85,B 0,C 180,E1 -21887.672,E2 -21887.672} C_VEL
LIN {X 0,Y 114.418,Z 689.908,A -85,B 0,C 180,E1 -21884.223,E2 -21884.223} C_VEL
LIN {X 0,Y 113.43,Z 691.284,A -85,B 0,C 180,E1 -21880.712,E2 -21880.712} C_VEL
LIN {X 0,Y 112.747,Z 692.256,A -85,B 0,C 180,E1 -21877.162,E2 -21877.162} C_VEL
LIN {X 0,Y 112.357,Z 692.847,A -85,B 0,C 180,E1 -21873.586,E2 -21873.586} C_VEL
LIN {X 0,Y 112.306,Z 693.045,A -85,B 0,C 180,E1 -21870,E2 -21870} C_VEL
LIN {X 0,Y 112.747,Z 692.209,A -85,B 0,C 180,E1 -21862.838,E2 -21862.838} C_VEL
LIN {X 0,Y 113.431,Z 691.218,A -85,B 0,C 180,E1 -21859.288,E2 -21859.288} C_VEL
LIN {X 0,Y 114.423,Z 689.805,A -85,B 0,C 180,E1 -21855.778,E2 -21855.778} C_VEL
LIN {X 0,Y 116.561,Z 686.877,A -85,B 0,C 180,E1 -21850.633,E2 -21850.633} C_VEL
LIN {X 0,Y 119.56,Z 682.898,A -85,B 0,C 180,E1 -21845.702,E2 -21845.702} C_VEL
LIN {X 0,Y 123.326,Z 677.752,A -85,B 0,C 180,E1 -21841.027,E2 -21841.027} C_VEL
LIN {X 0,Y 127.861,Z 671.272,A -85,B 0,C 180,E1 -21836.656,E2 -21836.656} C_VEL
LIN {X 0,Y 132.34,Z 664.203,A -85,B 0,C 180,E1 -21833.01,E2 -21833.01} C_VEL
LIN {X 0,Y 137.597,Z 654.937,A -85,B 0,C 180,E1 -21829.365,E2 -21829.365} C_VEL
LIN {X 0,Y 142.705,Z 644.713,A -85,B 0,C 180,E1 -21826.411,E2 -21826.411} C_VEL
LIN {X 0,Y 147.549,Z 633.227,A -85,B 0,C 180,E1 -21823.91,E2 -21823.91} C_VEL
LIN {X 0,Y 151.48,Z 621.7,A -85,B 0,C 180,E1 -21822.069,E2 -21822.069} C_VEL
LIN {X 0,Y 154.967,Z 608.6,A -85,B 0,C 180,E1 -21820.567,E2 -21820.567} C_VEL
LIN {X 0,Y 157.377,Z 595.989,A -85,B 0,C 180,E1 -21819.611,E2 -21819.611} C_VEL
LIN {X 0,Y 159.006,Z 581.209,A -85,B 0,C 180,E1 -21818.94,E2 -21818.94} C_VEL
LIN {X 0,Y 162.412,Z 536.201,A -85,B 0,C 180,E1 -21817.288,E2 -21817.288} C_VEL
LIN {X 0,Y 159.005,Z 527.506,A -85,B 0,C 180,E1 -21814.97,E2 -21814.97} C_VEL
LIN {X 0,Y 155.916,Z 520.75,A -85,B 0,C 180,E1 -21812.746,E2 -21812.746} C_VEL
LIN {X 0,Y 155.696,Z 520.593,A -85,B 0,C 180,E1 -21812.606,E2 -21812.606} C_VEL
LIN {X 0,Y 152.137,Z 531.074,A -85,B 0,C 180,E1 -21811.385,E2 -21811.385} C_VEL
LIN {X 0,Y 149.184,Z 538.086,A -85,B 0,C 180,E1 -21810.134,E2 -21810.134} C_VEL
LIN {X 0,Y 146.529,Z 542.77,A -85,B 0,C 180,E1 -21808.76,E2 -21808.76} C_VEL
LIN {X 0,Y 145.681,Z 544.197,A -85,B 0,C 180,E1 -21808.29,E2 -21808.29} C_VEL
LIN {X 0,Y 142.179,Z 556.642,A -85,B 0,C 180,E1 -21806.932,E2 -21806.932} C_VEL
LIN {X 0,Y 139.292,Z 565.107,A -85,B 0,C 180,E1 -21805.496,E2 -21805.496} C_VEL
LIN {X 0,Y 136.695,Z 571.343,A -85,B 0,C 180,E1 -21803.906,E2 -21803.906} C_VEL
LIN {X 0,Y 134.578,Z 575.464,A -85,B 0,C 180,E1 -21802.349,E2 -21802.349} C_VEL
LIN {X 0,Y 132.602,Z 578.055,A -85,B 0,C 180,E1 -21800.557,E2 -21800.557} C_VEL
LIN {X 0,Y 129.277,Z 588.289,A -85,B 0,C 180,E1 -21798.113,E2 -21798.113} C_VEL
LIN {X 0,Y 126.21,Z 595.945,A -85,B 0,C 180,E1 -21795.648,E2 -21795.648} C_VEL
LIN {X 0,Y 123.381,Z 601.648,A -85,B 0,C 180,E1 -21792.94,E2 -21792.94} C_VEL
LIN {X 0,Y 121.695,Z 604.415,A -85,B 0,C 180,E1 -21790.733,E2 -21790.733} C_VEL
LIN {X 0,Y 120.9,Z 605.244,A -85,B 0,C 180,E1 -21789.199,E2 -21789.199} C_VEL
LIN {X 0,Y 120.505,Z 605.605,A -85,B 0,C 180,E1 -21788.278,E2 -21788.278} C_VEL
LIN {X 0,Y 118.492,Z 610.295,A -85,B 0,C 180,E1 -21785.958,E2 -21785.958} C_VEL
LIN {X 0,Y 116.328,Z 615.136,A -85,B 0,C 180,E1 -21782.597,E2 -21782.597} C_VEL
LIN {X 0,Y 115.225,Z 617.751,A -85,B 0,C 180,E1 -21780,E2 -21780} C_VEL
LIN {X 0,Y 115.343,Z 618.44,A -85,B 0,C 180,E1 -21776.288,E2 -21776.288} C_VEL
LIN {X 0,Y 116.185,Z 628.009,A -85,B 0,C 180,E1 -21770.425,E2 -21770.425} C_VEL
LIN {X 0,Y 118.414,Z 636.309,A -85,B 0,C 180,E1 -21764.51,E2 -21764.51} C_VEL
LIN {X 0,Y 122.513,Z 644.091,A -85,B 0,C 180,E1 -21758.107,E2 -21758.107} C_VEL
LIN {X 0,Y 128.294,Z 650.329,A -85,B 0,C 180,E1 -21752.249,E2 -21752.249} C_VEL
LIN {X 0,Y 135.708,Z 655.242,A -85,B 0,C 180,E1 -21747.059,E2 -21747.059} C_VEL
LIN {X 0,Y 142.213,Z 658.09,A -85,B 0,C 180,E1 -21743.628,E2 -21743.628} C_VEL
LIN {X 0,Y 151.852,Z 660.782,A -85,B 0,C 180,E1 -21739.613,E2 -21739.613} C_VEL
LIN {X 0,Y 154.42,Z 661.283,A -85,B 0,C 180,E1 -21738.718,E2 -21738.718} C_VEL
LIN {X 0,Y 153.806,Z 661.539,A -85,B 0,C 180,E1 -21737.932,E2 -21737.932} C_VEL
LIN {X 0,Y 142.739,Z 661.792,A -85,B 0,C 180,E1 -21733.576,E2 -21733.576} C_VEL
LIN {X 0,Y 136.588,Z 661.499,A -85,B 0,C 180,E1 -21730.391,E2 -21730.391} C_VEL
LIN {X 0,Y 131.791,Z 668.732,A -85,B 0,C 180,E1 -21727.826,E2 -21727.826} C_VEL
LIN {X 0,Y 126.437,Z 676.884,A -85,B 0,C 180,E1 -21723.769,E2 -21723.769} C_VEL
LIN {X 0,Y 122.101,Z 683.45,A -85,B 0,C 180,E1 -21719.291,E2 -21719.291} C_VEL
LIN {X 0,Y 118.39,Z 688.67,A -85,B 0,C 180,E1 -21714.554,E2 -21714.554} C_VEL
LIN {X 0,Y 115.482,Z 692.712,A -85,B 0,C 180,E1 -21709.556,E2 -21709.556} C_VEL
LIN {X 0,Y 113.623,Z 695.701,A -85,B 0,C 180,E1 -21704.325,E2 -21704.325} C_VEL
LIN {X 0,Y 112.786,Z 697.145,A -85,B 0,C 180,E1 -21700.774,E2 -21700.774} C_VEL
LIN {X 0,Y 112.334,Z 698.164,A -85,B 0,C 180,E1 -21697.188,E2 -21697.188} C_VEL
LIN {X 0,Y 112.182,Z 698.792,A -85,B 0,C 180,E1 -21693.592,E2 -21693.592} C_VEL
LIN {X 0,Y 112.305,Z 699.028,A -85,B 0,C 180,E1 -21690,E2 -21690} C_VEL
LIN {X 0,Y 112.272,Z 698.811,A -85,B 0,C 180,E1 -21686.411,E2 -21686.411} C_VEL
LIN {X 0,Y 113.086,Z 697.191,A -85,B 0,C 180,E1 -21679.255,E2 -21679.255} C_VEL
LIN {X 0,Y 114.132,Z 695.776,A -85,B 0,C 180,E1 -21675.741,E2 -21675.741} C_VEL
LIN {X 0,Y 116.533,Z 692.825,A -85,B 0,C 180,E1 -21670.628,E2 -21670.628} C_VEL
LIN {X 0,Y 120.022,Z 688.83,A -85,B 0,C 180,E1 -21665.802,E2 -21665.802} C_VEL
LIN {X 0,Y 122.191,Z 686.564,A -85,B 0,C 180,E1 -21663.528,E2 -21663.528} C_VEL
LIN {X 0,Y 125.444,Z 689.166,A -85,B 0,C 180,E1 -21659.72,E2 -21659.72} C_VEL
LIN {X 0,Y 131.977,Z 692.316,A -85,B 0,C 180,E1 -21654.142,E2 -21654.142} C_VEL
LIN {X 0,Y 140.257,Z 694.49,A -85,B 0,C 180,E1 -21649.352,E2 -21649.352} C_VEL
LIN {X 0,Y 149.837,Z 695.632,A -85,B 0,C 180,E1 -21645.286,E2 -21645.286} C_VEL
LIN {X 0,Y 152.263,Z 695.668,A -85,B 0,C 180,E1 -21643.817,E2 -21643.817} C_VEL
LIN {X 0,Y 142.545,Z 694.013,A -85,B 0,C 180,E1 -21639.863,E2 -21639.863} C_VEL
LIN {X 0,Y 133.935,Z 691.235,A -85,B 0,C 180,E1 -21635.254,E2 -21635.254} C_VEL
LIN {X 0,Y 126.809,Z 687.309,A -85,B 0,C 180,E1 -21629.92,E2 -21629.92} C_VEL
LIN {X 0,Y 121.47,Z 682.228,A -85,B 0,C 180,E1 -21623.891,E2 -21623.891} C_VEL
LIN {X 0,Y 117.726,Z 675.078,A -85,B 0,C 180,E1 -21616.655,E2 -21616.655} C_VEL
LIN {X 0,Y 116.277,Z 667.753,A -85,B 0,C 180,E1 -21610.447,E2 -21610.447} C_VEL
LIN {X 0,Y 116.156,Z 661.769,A -85,B 0,C 180,E1 -21606.078,E2 -21606.078} C_VEL
LIN {X 0,Y 116.132,Z 654.46,A -85,B 0,C 180,E1 -21601.734,E2 -21601.734} C_VEL
LIN {X 0,Y 116.198,Z 645.615,A -85,B 0,C 180,E1 -21597.4,E2 -21597.4} C_VEL
LIN {X 0,Y 116.47,Z 635.946,A -85,B 0,C 180,E1 -21593.503,E2 -21593.503} C_VEL
LIN {X 0,Y 116.549,Z 634.295,A -85,B 0,C 180,E1 -21592.916,E2 -21592.916} C_VEL
LIN {X 0,Y 116.433,Z 631.544,A -85,B 0,C 180,E1 -21591.515,E2 -21591.515} C_VEL
LIN {X 0,Y 115.922,Z 629.628,A -85,B 0,C 180,E1 -21589.777,E2 -21589.777} C_VEL
LIN {X 0,Y 115.432,Z 627.095,A -85,B 0,C 180,E1 -21585.885,E2 -21585.885} C_VEL
LIN {X 0,Y 116.241,Z 625.796,A -85,B 0,C 180,E1 -21584.001,E2 -21584.001} C_VEL
LIN {X 0,Y 116.763,Z 625.281,A -85,B 0,C 180,E1 -21583.434,E2 -21583.434} C_VEL
LIN {X 0,Y 118.592,Z 623.408,A -85,B 0,C 180,E1 -21581.963,E2 -21581.963} C_VEL
LIN {X 0,Y 121.825,Z 619.185,A -85,B 0,C 180,E1 -21580.189,E2 -21580.189} C_VEL
LIN {X 0,Y 122.518,Z 618.13,A -85,B 0,C 180,E1 -21579.868,E2 -21579.868} C_VEL
LIN {X 0,Y 125.201,Z 615.95,A -85,B 0,C 180,E1 -21577.734,E2 -21577.734} C_VEL
LIN {X 0,Y 128.503,Z 612.057,A -85,B 0,C 180,E1 -21575.874,E2 -21575.874} C_VEL
LIN {X 0,Y 132.243,Z 606.133,A -85,B 0,C 180,E1 -21574.335,E2 -21574.335} C_VEL
LIN {X 0,Y 135.796,Z 598.75,A -85,B 0,C 180,E1 -21573.178,E2 -21573.178} C_VEL
LIN {X 0,Y 137.537,Z 594.34,A -85,B 0,C 180,E1 -21572.62,E2 -21572.62} C_VEL
LIN {X 0,Y 140.378,Z 590.131,A -85,B 0,C 180,E1 -21571.09,E2 -21571.09} C_VEL
LIN {X 0,Y 143.252,Z 584.139,A -85,B 0,C 180,E1 -21569.757,E2 -21569.757} C_VEL
LIN {X 0,Y 146.813,Z 574.393,A -85,B 0,C 180,E1 -21568.331,E2 -21568.331} C_VEL
LIN {X 0,Y 150.645,Z 561.883,A -85,B 0,C 180,E1 -21567.1,E2 -21567.1} C_VEL
LIN {X 0,Y 153.808,Z 556.912,A -85,B 0,C 180,E1 -21565.72,E2 -21565.72} C_VEL
LIN {X 0,Y 157.393,Z 549.32,A -85,B 0,C 180,E1 -21564.427,E2 -21564.427} C_VEL
LIN {X 0,Y 153.986,Z 589.817,A -85,B 0,C 180,E1 -21562.94,E2 -21562.94} C_VEL
LIN {X 0,Y 151.936,Z 602.799,A -85,B 0,C 180,E1 -21562.159,E2 -21562.159} C_VEL
LIN {X 0,Y 148.925,Z 615.766,A -85,B 0,C 180,E1 -21560.87,E2 -21560.87} C_VEL
LIN {X 0,Y 145.578,Z 626.267,A -85,B 0,C 180,E1 -21559.496,E2 -21559.496} C_VEL
LIN {X 0,Y 140.951,Z 638.188,A -85,B 0,C 180,E1 -21557.346,E2 -21557.346} C_VEL
LIN {X 0,Y 135.946,Z 648.701,A -85,B 0,C 180,E1 -21554.779,E2 -21554.779} C_VEL
LIN {X 0,Y 131.165,Z 657.302,A -85,B 0,C 180,E1 -21552.049,E2 -21552.049} C_VEL
LIN {X 0,Y 126.082,Z 665.68,A -85,B 0,C 180,E1 -21548.496,E2 -21548.496} C_VEL
LIN {X 0,Y 121.133,Z 672.936,A -85,B 0,C 180,E1 -21544.45,E2 -21544.45} C_VEL
LIN {X 0,Y 117.151,Z 678.173,A -85,B 0,C 180,E1 -21540.659,E2 -21540.659} C_VEL
LIN {X 0,Y 113.051,Z 683.275,A -85,B 0,C 180,E1 -21535.796,E2 -21535.796} C_VEL
LIN {X 0,Y 109.866,Z 687.207,A -85,B 0,C 180,E1 -21530.599,E2 -21530.599} C_VEL
LIN {X 0,Y 107.553,Z 690.096,A -85,B 0,C 180,E1 -21525.152,E2 -21525.152} C_VEL
LIN {X 0,Y 106.453,Z 691.472,A -85,B 0,C 180,E1 -21521.424,E2 -21521.424} C_VEL
LIN {X 0,Y 105.716,Z 692.445,A -85,B 0,C 180,E1 -21517.641,E2 -21517.641} C_VEL
LIN {X 0,Y 105.225,Z 693.234,A -85,B 0,C 180,E1 -21510,E2 -21510} C_VEL
LIN {X 0,Y 105.716,Z 692.398,A -85,B 0,C 180,E1 -21502.359,E2 -21502.359} C_VEL
LIN {X 0,Y 106.454,Z 691.408,A -85,B 0,C 180,E1 -21498.577,E2 -21498.577} C_VEL
LIN {X 0,Y 107.558,Z 689.994,A -85,B 0,C 180,E1 -21494.849,E2 -21494.849} C_VEL
LIN {X 0,Y 109.887,Z 687.067,A -85,B 0,C 180,E1 -21489.405,E2 -21489.405} C_VEL
LIN {X 0,Y 113.105,Z 683.088,A -85,B 0,C 180,E1 -21484.217,E2 -21484.217} C_VEL
LIN {X 0,Y 117.172,Z 677.94,A -85,B 0,C 180,E1 -21479.347,E2 -21479.347} C_VEL
LIN {X 0,Y 121.989,Z 671.46,A -85,B 0,C 180,E1 -21474.822,E2 -21474.822} C_VEL
LIN {X 0,Y 127.499,Z 663.181,A -85,B 0,C 180,E1 -21470.508,E2 -21470.508} C_VEL
LIN {X 0,Y 132.293,Z 655.123,A -85,B 0,C 180,E1 -21467.364,E2 -21467.364} C_VEL
LIN {X 0,Y 137.658,Z 644.896,A -85,B 0,C 180,E1 -21464.376,E2 -21464.376} C_VEL
LIN {X 0,Y 142.722,Z 633.407,A -85,B 0,C 180,E1 -21461.858,E2 -21461.858} C_VEL
LIN {X 0,Y 146.818,Z 621.875,A -85,B 0,C 180,E1 -21460.013,E2 -21460.013} C_VEL
LIN {X 0,Y 150.436,Z 608.767,A -85,B 0,C 180,E1 -21458.508,E2 -21458.508} C_VEL
LIN {X 0,Y 153.023,Z 595.674,A -85,B 0,C 180,E1 -21457.54,E2 -21457.54} C_VEL
LIN {X 0,Y 154.64,Z 581.446,A -85,B 0,C 180,E1 -21456.903,E2 -21456.903} C_VEL
LIN {X 0,Y 158.019,Z 538.627,A -85,B 0,C 180,E1 -21455.323,E2 -21455.323} C_VEL
LIN {X 0,Y 155.992,Z 533.312,A -85,B 0,C 180,E1 -21453.825,E2 -21453.825} C_VEL
LIN {X 0,Y 155.52,Z 533.421,A -85,B 0,C 180,E1 -21453.572,E2 -21453.572} C_VEL
LIN {X 0,Y 151.981,Z 541.68,A -85,B 0,C 180,E1 -21452.225,E2 -21452.225} C_VEL
LIN {X 0,Y 148.855,Z 547.207,A -85,B 0,C 180,E1 -21450.771,E2 -21450.771} C_VEL
LIN {X 0,Y 148.275,Z 548.08,A -85,B 0,C 180,E1 -21450.473,E2 -21450.473} C_VEL
LIN {X 0,Y 144.831,Z 559.745,A -85,B 0,C 180,E1 -21449.248,E2 -21449.248} C_VEL
LIN {X 0,Y 141.725,Z 568.45,A -85,B 0,C 180,E1 -21447.854,E2 -21447.854} C_VEL
LIN {X 0,Y 138.729,Z 575.372,A -85,B 0,C 180,E1 -21446.212,E2 -21446.212} C_VEL
LIN {X 0,Y 135.897,Z 580.67,A -85,B 0,C 180,E1 -21444.338,E2 -21444.338} C_VEL
LIN {X 0,Y 133.826,Z 583.564,A -85,B 0,C 180,E1 -21442.685,E2 -21442.685} C_VEL
LIN {X 0,Y 129.866,Z 593.995,A -85,B 0,C 180,E1 -21440.182,E2 -21440.182} C_VEL
LIN {X 0,Y 125.832,Z 602.208,A -85,B 0,C 180,E1 -21437.438,E2 -21437.438} C_VEL
LIN {X 0,Y 122.296,Z 608.028,A -85,B 0,C 180,E1 -21434.455,E2 -21434.455} C_VEL
LIN {X 0,Y 120.181,Z 610.826,A -85,B 0,C 180,E1 -21431.983,E2 -21431.983} C_VEL
LIN {X 0,Y 119.129,Z 611.807,A -85,B 0,C 180,E1 -21430.194,E2 -21430.194} C_VEL
LIN {X 0,Y 116.046,Z 617.494,A -85,B 0,C 180,E1 -21426.957,E2 -21426.957} C_VEL
LIN {X 0,Y 113.687,Z 621.785,A -85,B 0,C 180,E1 -21423.544,E2 -21423.544} C_VEL
LIN {X 0,Y 112.743,Z 623.573,A -85,B 0,C 180,E1 -21421.608,E2 -21421.608} C_VEL
LIN {X 0,Y 111.787,Z 626.278,A -85,B 0,C 180,E1 -21416.396,E2 -21416.396} C_VEL
LIN {X 0,Y 110.507,Z 630.291,A -85,B 0,C 180,E1 -21412.693,E2 -21412.693} C_VEL
LIN {X 0,Y 110.126,Z 633.231,A -85,B 0,C 180,E1 -21408.963,E2 -21408.963} C_VEL
LIN {X 0,Y 110.8,Z 635.018,A -85,B 0,C 180,E1 -21405.302,E2 -21405.302} C_VEL
LIN {X 0,Y 111.989,Z 635.139,A -85,B 0,C 180,E1 -21403.127,E2 -21403.127} C_VEL
LIN {X 0,Y 112.308,Z 635.203,A -85,B 0,C 180,E1 -21402.708,E2 -21402.708} C_VEL
LIN {X 0,Y 116.131,Z 642.343,A -85,B 0,C 180,E1 -21396.836,E2 -21396.836} C_VEL
LIN {X 0,Y 122.155,Z 649.078,A -85,B 0,C 180,E1 -21390.723,E2 -21390.723} C_VEL
LIN {X 0,Y 129.834,Z 654.488,A -85,B 0,C 180,E1 -21385.363,E2 -21385.363} C_VEL
LIN {X 0,Y 136.564,Z 657.708,A -85,B 0,C 180,E1 -21381.862,E2 -21381.862} C_VEL
LIN {X 0,Y 143.126,Z 660.011,A -85,B 0,C 180,E1 -21379.074,E2 -21379.074} C_VEL
LIN {X 0,Y 143.685,Z 660.495,A -85,B 0,C 180,E1 -21378.001,E2 -21378.001} C_VEL
LIN {X 0,Y 132.381,Z 659.73,A -85,B 0,C 180,E1 -21372.86,E2 -21372.86} C_VEL
LIN {X 0,Y 127.339,Z 666.99,A -85,B 0,C 180,E1 -21370.429,E2 -21370.429} C_VEL
LIN {X 0,Y 122.323,Z 674.181,A -85,B 0,C 180,E1 -21367.105,E2 -21367.105} C_VEL
LIN {X 0,Y 117.421,Z 681.253,A -85,B 0,C 180,E1 -21362.594,E2 -21362.594} C_VEL
LIN {X 0,Y 113.152,Z 686.871,A -85,B 0,C 180,E1 -21357.764,E2 -21357.764} C_VEL
LIN {X 0,Y 109.721,Z 691.283,A -85,B 0,C 180,E1 -21352.602,E2 -21352.602} C_VEL
LIN {X 0,Y 107.981,Z 693.61,A -85,B 0,C 180,E1 -21348.992,E2 -21348.992} C_VEL
LIN {X 0,Y 106.711,Z 695.511,A -85,B 0,C 180,E1 -21345.274,E2 -21345.274} C_VEL
LIN {X 0,Y 105.805,Z 696.955,A -85,B 0,C 180,E1 -21341.494,E2 -21341.494} C_VEL
LIN {X 0,Y 105.277,Z 697.974,A -85,B 0,C 180,E1 -21337.673,E2 -21337.673} C_VEL
LIN {X 0,Y 105.098,Z 698.603,A -85,B 0,C 180,E1 -21333.834,E2 -21333.834} C_VEL
LIN {X 0,Y 105.221,Z 698.839,A -85,B 0,C 180,E1 -21330,E2 -21330} C_VEL
LIN {X 0,Y 105.192,Z 698.623,A -85,B 0,C 180,E1 -21326.169,E2 -21326.169} C_VEL
LIN {X 0,Y 106.13,Z 697.003,A -85,B 0,C 180,E1 -21318.541,E2 -21318.541} C_VEL
LIN {X 0,Y 107.259,Z 695.587,A -85,B 0,C 180,E1 -21314.805,E2 -21314.805} C_VEL
LIN {X 0,Y 109.857,Z 692.638,A -85,B 0,C 180,E1 -21309.399,E2 -21309.399} C_VEL
LIN {X 0,Y 113.595,Z 688.643,A -85,B 0,C 180,E1 -21304.337,E2 -21304.337} C_VEL
LIN {X 0,Y 117.088,Z 685.063,A -85,B 0,C 180,E1 -21300.934,E2 -21300.934} C_VEL
LIN {X 0,Y 122.869,Z 688.968,A -85,B 0,C 180,E1 -21295.11,E2 -21295.11} C_VEL
LIN {X 0,Y 130.558,Z 692.041,A -85,B 0,C 180,E1 -21289.762,E2 -21289.762} C_VEL
LIN {X 0,Y 139.842,Z 694.165,A -85,B 0,C 180,E1 -21285.284,E2 -21285.284} C_VEL
LIN {X 0,Y 142.099,Z 694.426,A -85,B 0,C 180,E1 -21283.822,E2 -21283.822} C_VEL
LIN {X 0,Y 132.596,Z 691.728,A -85,B 0,C 180,E1 -21279.497,E2 -21279.497} C_VEL
LIN {X 0,Y 124.368,Z 687.915,A -85,B 0,C 180,E1 -21274.409,E2 -21274.409} C_VEL
LIN {X 0,Y 117.901,Z 682.984,A -85,B 0,C 180,E1 -21268.481,E2 -21268.481} C_VEL
LIN {X 0,Y 113.209,Z 676.796,A -85,B 0,C 180,E1 -21261.868,E2 -21261.868} C_VEL
LIN {X 0,Y 110.587,Z 669.21,A -85,B 0,C 180,E1 -21254.726,E2 -21254.726} C_VEL
LIN {X 0,Y 109.825,Z 659.71,A -85,B 0,C 180,E1 -21247.353,E2 -21247.353} C_VEL
LIN {X 0,Y 109.684,Z 652.274,A -85,B 0,C 180,E1 -21242.754,E2 -21242.754} C_VEL
LIN {X 0,Y 109.72,Z 641.996,A -85,B 0,C 180,E1 -21237.705,E2 -21237.705} C_VEL
LIN {X 0,Y 109.976,Z 631.012,A -85,B 0,C 180,E1 -21233.233,E2 -21233.233} C_VEL
LIN {X 0,Y 109.613,Z 631.868,A -85,B 0,C 180,E1 -21232.632,E2 -21232.632} C_VEL
LIN {X 0,Y 111.29,Z 630.706,A -85,B 0,C 180,E1 -21229.079,E2 -21229.079} C_VEL
LIN {X 0,Y 113.185,Z 628.316,A -85,B 0,C 180,E1 -21227.448,E2 -21227.448} C_VEL
LIN {X 0,Y 114.679,Z 626.866,A -85,B 0,C 180,E1 -21225.81,E2 -21225.81} C_VEL
LIN {X 0,Y 115.969,Z 626.015,A -85,B 0,C 180,E1 -21224.174,E2 -21224.174} C_VEL
LIN {X 0,Y 116.763,Z 625.281,A -85,B 0,C 180,E1 -21223.434,E2 -21223.434} C_VEL
LIN {X 0,Y 118.973,Z 623.782,A -85,B 0,C 180,E1 -21221.156,E2 -21221.156} C_VEL
LIN {X 0,Y 123.808,Z 621.72,A -85,B 0,C 180,E1 -21216.357,E2 -21216.357} C_VEL
LIN {X 0,Y 126.248,Z 619.763,A -85,B 0,C 180,E1 -21214.812,E2 -21214.812} C_VEL
LIN {X 0,Y 129.293,Z 616.372,A -85,B 0,C 180,E1 -21213.393,E2 -21213.393} C_VEL
LIN {X 0,Y 133.902,Z 609.725,A -85,B 0,C 180,E1 -21211.811,E2 -21211.811} C_VEL
LIN {X 0,Y 137.929,Z 602.134,A -85,B 0,C 180,E1 -21210.706,E2 -21210.706} C_VEL
LIN {X 0,Y 139.571,Z 598.55,A -85,B 0,C 180,E1 -21210.269,E2 -21210.269} C_VEL
LIN {X 0,Y 143.187,Z 593.3,A -85,B 0,C 180,E1 -21208.67,E2 -21208.67} C_VEL
LIN {X 0,Y 146.737,Z 585.965,A -85,B 0,C 180,E1 -21207.319,E2 -21207.319} C_VEL
LIN {X 0,Y 150.418,Z 576.022,A -85,B 0,C 180,E1 -21206.029,E2 -21206.029} C_VEL
LIN {X 0,Y 151.371,Z 573.133,A -85,B 0,C 180,E1 -21205.735,E2 -21205.735} C_VEL
LIN {X 0,Y 149.473,Z 592.597,A -85,B 0,C 180,E1 -21204.983,E2 -21204.983} C_VEL
LIN {X 0,Y 147.013,Z 606.07,A -85,B 0,C 180,E1 -21204.067,E2 -21204.067} C_VEL
LIN {X 0,Y 143.937,Z 618.091,A -85,B 0,C 180,E1 -21202.797,E2 -21202.797} C_VEL
LIN {X 0,Y 140.467,Z 628.141,A -85,B 0,C 180,E1 -21201.423,E2 -21201.423} C_VEL
LIN {X 0,Y 135.686,Z 639.62,A -85,B 0,C 180,E1 -21199.246,E2 -21199.246} C_VEL
LIN {X 0,Y 130.421,Z 649.924,A -85,B 0,C 180,E1 -21196.676,E2 -21196.676} C_VEL
LIN {X 0,Y 124.931,Z 659.22,A -85,B 0,C 180,E1 -21193.561,E2 -21193.561} C_VEL
LIN {X 0,Y 118.978,Z 668.14,A -85,B 0,C 180,E1 -21189.42,E2 -21189.42} C_VEL
LIN {X 0,Y 113.593,Z 675.319,A -85,B 0,C 180,E1 -21184.911,E2 -21184.911} C_VEL
LIN {X 0,Y 109.518,Z 680.178,A -85,B 0,C 180,E1 -21180.889,E2 -21180.889} C_VEL
LIN {X 0,Y 105.468,Z 684.871,A -85,B 0,C 180,E1 -21175.667,E2 -21175.667} C_VEL
LIN {X 0,Y 102.291,Z 688.446,A -85,B 0,C 180,E1 -21170.092,E2 -21170.092} C_VEL
LIN {X 0,Y 100.703,Z 690.284,A -85,B 0,C 180,E1 -21166.21,E2 -21166.21} C_VEL
LIN {X 0,Y 99.51,Z 691.661,A -85,B 0,C 180,E1 -21162.233,E2 -21162.233} C_VEL
LIN {X 0,Y 98.682,Z 692.634,A -85,B 0,C 180,E1 -21158.189,E2 -21158.189} C_VEL
LIN {X 0,Y 98.216,Z 693.224,A -85,B 0,C 180,E1 -21154.103,E2 -21154.103} C_VEL
LIN {X 0,Y 98.145,Z 693.423,A -85,B 0,C 180,E1 -21150,E2 -21150} C_VEL
LIN {X 0,Y 98.683,Z 692.588,A -85,B 0,C 180,E1 -21141.811,E2 -21141.811} C_VEL
LIN {X 0,Y 99.511,Z 691.597,A -85,B 0,C 180,E1 -21137.768,E2 -21137.768} C_VEL
LIN {X 0,Y 100.709,Z 690.184,A -85,B 0,C 180,E1 -21133.791,E2 -21133.791} C_VEL
LIN {X 0,Y 103.276,Z 687.256,A -85,B 0,C 180,E1 -21128.02,E2 -21128.02} C_VEL
LIN {X 0,Y 106.737,Z 683.278,A -85,B 0,C 180,E1 -21122.554,E2 -21122.554} C_VEL
LIN {X 0,Y 111.13,Z 678.129,A -85,B 0,C 180,E1 -21117.483,E2 -21117.483} C_VEL
LIN {X 0,Y 116.256,Z 671.648,A -85,B 0,C 180,E1 -21112.805,E2 -21112.805} C_VEL
LIN {X 0,Y 122.263,Z 663.115,A -85,B 0,C 180,E1 -21108.267,E2 -21108.267} C_VEL
LIN {X 0,Y 128.241,Z 653.407,A -85,B 0,C 180,E1 -21104.566,E2 -21104.566} C_VEL
LIN {X 0,Y 133.946,Z 642.787,A -85,B 0,C 180,E1 -21101.61,E2 -21101.61} C_VEL
LIN {X 0,Y 138.694,Z 632.078,A -85,B 0,C 180,E1 -21099.397,E2 -21099.397} C_VEL
LIN {X 0,Y 143.017,Z 620.131,A -85,B 0,C 180,E1 -21097.59,E2 -21097.59} C_VEL
LIN {X 0,Y 146.43,Z 607.62,A -85,B 0,C 180,E1 -21096.203,E2 -21096.203} C_VEL
LIN {X 0,Y 148.992,Z 594.626,A -85,B 0,C 180,E1 -21095.308,E2 -21095.308} C_VEL
LIN {X 0,Y 150.613,Z 580.3,A -85,B 0,C 180,E1 -21094.709,E2 -21094.709} C_VEL
LIN {X 0,Y 153.153,Z 548.68,A -85,B 0,C 180,E1 -21093.506,E2 -21093.506} C_VEL
LIN {X 0,Y 150.992,Z 552.335,A -85,B 0,C 180,E1 -21092.56,E2 -21092.56} C_VEL
LIN {X 0,Y 147.513,Z 563.442,A -85,B 0,C 180,E1 -21091.406,E2 -21091.406} C_VEL
LIN {X 0,Y 144.114,Z 572.424,A -85,B 0,C 180,E1 -21090.001,E2 -21090.001} C_VEL
LIN {X 0,Y 140.748,Z 579.837,A -85,B 0,C 180,E1 -21088.318,E2 -21088.318} C_VEL
LIN {X 0,Y 137.255,Z 585.997,A -85,B 0,C 180,E1 -21086.208,E2 -21086.208} C_VEL
LIN {X 0,Y 135.171,Z 588.924,A -85,B 0,C 180,E1 -21084.784,E2 -21084.784} C_VEL
LIN {X 0,Y 130.84,Z 598.683,A -85,B 0,C 180,E1 -21082.502,E2 -21082.502} C_VEL
LIN {X 0,Y 126.057,Z 607.097,A -85,B 0,C 180,E1 -21079.776,E2 -21079.776} C_VEL
LIN {X 0,Y 121.842,Z 613.134,A -85,B 0,C 180,E1 -21076.763,E2 -21076.763} C_VEL
LIN {X 0,Y 120.173,Z 615.222,A -85,B 0,C 180,E1 -21075.258,E2 -21075.258} C_VEL
LIN {X 0,Y 118.274,Z 617.159,A -85,B 0,C 180,E1 -21073.085,E2 -21073.085} C_VEL
LIN {X 0,Y 117.573,Z 617.789,A -85,B 0,C 180,E1 -21072.077,E2 -21072.077} C_VEL
LIN {X 0,Y 113.679,Z 623.789,A -85,B 0,C 180,E1 -21068.437,E2 -21068.437} C_VEL
LIN {X 0,Y 111.314,Z 627.317,A -85,B 0,C 180,E1 -21065.435,E2 -21065.435} C_VEL
LIN {X 0,Y 110.257,Z 628.934,A -85,B 0,C 180,E1 -21063.655,E2 -21063.655} C_VEL
LIN {X 0,Y 108.671,Z 631.866,A -85,B 0,C 180,E1 -21058.147,E2 -21058.147} C_VEL
LIN {X 0,Y 107.081,Z 635.651,A -85,B 0,C 180,E1 -21054.35,E2 -21054.35} C_VEL
LIN {X 0,Y 106.494,Z 637.605,A -85,B 0,C 180,E1 -21051.857,E2 -21051.857} C_VEL
LIN {X 0,Y 106.396,Z 639.558,A -85,B 0,C 180,E1 -21048.57,E2 -21048.57} C_VEL
LIN {X 0,Y 108.343,Z 642.636,A -85,B 0,C 180,E1 -21041.075,E2 -21041.075} C_VEL
LIN {X 0,Y 109.425,Z 644.996,A -85,B 0,C 180,E1 -21037.334,E2 -21037.334} C_VEL
LIN {X 0,Y 111.364,Z 646.667,A -85,B 0,C 180,E1 -21033.784,E2 -21033.784} C_VEL
LIN {X 0,Y 114.246,Z 647.445,A -85,B 0,C 180,E1 -21030.519,E2 -21030.519} C_VEL
LIN {X 0,Y 116.152,Z 647.563,A -85,B 0,C 180,E1 -21029.049,E2 -21029.049} C_VEL
LIN {X 0,Y 124.103,Z 653.465,A -85,B 0,C 180,E1 -21023.515,E2 -21023.515} C_VEL
LIN {X 0,Y 133.87,Z 658.27,A -85,B 0,C 180,E1 -21018.719,E2 -21018.719} C_VEL
LIN {X 0,Y 133.11,Z 658.439,A -85,B 0,C 180,E1 -21017.662,E2 -21017.662} C_VEL
LIN {X 0,Y 128.499,Z 657.866,A -85,B 0,C 180,E1 -21015.457,E2 -21015.457} C_VEL
LIN {X 0,Y 123.198,Z 665.194,A -85,B 0,C 180,E1 -21013.201,E2 -21013.201} C_VEL
LIN {X 0,Y 117.73,Z 672.65,A -85,B 0,C 180,E1 -21009.921,E2 -21009.921} C_VEL
LIN {X 0,Y 112.545,Z 679.608,A -85,B 0,C 180,E1 -21005.642,E2 -21005.642} C_VEL
LIN {X 0,Y 108.335,Z 684.934,A -85,B 0,C 180,E1 -21001.264,E2 -21001.264} C_VEL
LIN {X 0,Y 104.328,Z 689.74,A -85,B 0,C 180,E1 -20995.968,E2 -20995.968} C_VEL
LIN {X 0,Y 101.249,Z 693.419,A -85,B 0,C 180,E1 -20990.308,E2 -20990.308} C_VEL
LIN {X 0,Y 99.834,Z 695.32,A -85,B 0,C 180,E1 -20986.355,E2 -20986.355} C_VEL
LIN {X 0,Y 98.82,Z 696.765,A -85,B 0,C 180,E1 -20982.319,E2 -20982.319} C_VEL
LIN {X 0,Y 98.245,Z 697.785,A -85,B 0,C 180,E1 -20978.226,E2 -20978.226} C_VEL
LIN {X 0,Y 98.013,Z 698.414,A -85,B 0,C 180,E1 -20974.112,E2 -20974.112} C_VEL
LIN {X 0,Y 98.139,Z 698.651,A -85,B 0,C 180,E1 -20970,E2 -20970} C_VEL
LIN {X 0,Y 98.106,Z 698.434,A -85,B 0,C 180,E1 -20965.892,E2 -20965.892} C_VEL
LIN {X 0,Y 99.174,Z 696.814,A -85,B 0,C 180,E1 -20957.725,E2 -20957.725} C_VEL
LIN {X 0,Y 100.427,Z 695.399,A -85,B 0,C 180,E1 -20953.744,E2 -20953.744} C_VEL
LIN {X 0,Y 103.246,Z 692.45,A -85,B 0,C 180,E1 -20948.013,E2 -20948.013} C_VEL
LIN {X 0,Y 107.235,Z 688.457,A -85,B 0,C 180,E1 -20942.692,E2 -20942.692} C_VEL
LIN {X 0,Y 112.504,Z 683.502,A -85,B 0,C 180,E1 -20937.928,E2 -20937.928} C_VEL
LIN {X 0,Y 117.376,Z 686.839,A -85,B 0,C 180,E1 -20933.219,E2 -20933.219} C_VEL
LIN {X 0,Y 125.389,Z 690.314,A -85,B 0,C 180,E1 -20927.732,E2 -20927.732} C_VEL
LIN {X 0,Y 130.022,Z 691.72,A -85,B 0,C 180,E1 -20925.357,E2 -20925.357} C_VEL
LIN {X 0,Y 132.063,Z 692.148,A -85,B 0,C 180,E1 -20923.774,E2 -20923.774} C_VEL
LIN {X 0,Y 122.869,Z 688.438,A -85,B 0,C 180,E1 -20918.99,E2 -20918.99} C_VEL
LIN {X 0,Y 115.15,Z 683.619,A -85,B 0,C 180,E1 -20913.319,E2 -20913.319} C_VEL
LIN {X 0,Y 109.334,Z 677.651,A -85,B 0,C 180,E1 -20906.741,E2 -20906.741} C_VEL
LIN {X 0,Y 105.859,Z 671.316,A -85,B 0,C 180,E1 -20900.359,E2 -20900.359} C_VEL
LIN {X 0,Y 103.806,Z 662.6,A -85,B 0,C 180,E1 -20892.711,E2 -20892.711} C_VEL
LIN {X 0,Y 103.549,Z 656.047,A -85,B 0,C 180,E1 -20887.801,E2 -20887.801} C_VEL
LIN {X 0,Y 103.395,Z 649.771,A -85,B 0,C 180,E1 -20883.897,E2 -20883.897} C_VEL
LIN {X 0,Y 103.253,Z 641.107,A -85,B 0,C 180,E1 -20879.39,E2 -20879.39} C_VEL
LIN {X 0,Y 102.628,Z 642.016,A -85,B 0,C 180,E1 -20878.038,E2 -20878.038} C_VEL
LIN {X 0,Y 102.98,Z 641.682,A -85,B 0,C 180,E1 -20876.087,E2 -20876.087} C_VEL
LIN {X 0,Y 104.824,Z 639.55,A -85,B 0,C 180,E1 -20873.262,E2 -20873.262} C_VEL
LIN {X 0,Y 105.711,Z 638.441,A -85,B 0,C 180,E1 -20872.359,E2 -20872.359} C_VEL
LIN {X 0,Y 108.957,Z 636.012,A -85,B 0,C 180,E1 -20866.952,E2 -20866.952} C_VEL
LIN {X 0,Y 111.038,Z 633.794,A -85,B 0,C 180,E1 -20865.334,E2 -20865.334} C_VEL
LIN {X 0,Y 115.611,Z 630.326,A -85,B 0,C 180,E1 -20860.928,E2 -20860.928} C_VEL
LIN {X 0,Y 118.429,Z 627.54,A -85,B 0,C 180,E1 -20859.141,E2 -20859.141} C_VEL
LIN {X 0,Y 121.576,Z 623.881,A -85,B 0,C 180,E1 -20857.657,E2 -20857.657} C_VEL
LIN {X 0,Y 125.533,Z 620.487,A -85,B 0,C 180,E1 -20855.172,E2 -20855.172} C_VEL
LIN {X 0,Y 126.248,Z 619.763,A -85,B 0,C 180,E1 -20854.812,E2 -20854.812} C_VEL
LIN {X 0,Y 135.015,Z 611.032,A -85,B 0,C 180,E1 -20850.594,E2 -20850.594} C_VEL
LIN {X 0,Y 140.323,Z 604.872,A -85,B 0,C 180,E1 -20848.393,E2 -20848.393} C_VEL
LIN {X 0,Y 143.277,Z 600.585,A -85,B 0,C 180,E1 -20847.353,E2 -20847.353} C_VEL
LIN {X 0,Y 144.393,Z 599.061,A -85,B 0,C 180,E1 -20846.946,E2 -20846.946} C_VEL
LIN {X 0,Y 141.811,Z 611.056,A -85,B 0,C 180,E1 -20845.901,E2 -20845.901} C_VEL
LIN {X 0,Y 138.065,Z 623.104,A -85,B 0,C 180,E1 -20844.534,E2 -20844.534} C_VEL
LIN {X 0,Y 133.653,Z 634.403,A -85,B 0,C 180,E1 -20842.687,E2 -20842.687} C_VEL
LIN {X 0,Y 128.053,Z 645.795,A -85,B 0,C 180,E1 -20840.208,E2 -20840.208} C_VEL
LIN {X 0,Y 122.124,Z 655.918,A -85,B 0,C 180,E1 -20837.201,E2 -20837.201} C_VEL
LIN {X 0,Y 115.695,Z 665.451,A -85,B 0,C 180,E1 -20833.201,E2 -20833.201} C_VEL
LIN {X 0,Y 109.708,Z 673.306,A -85,B 0,C 180,E1 -20828.653,E2 -20828.653} C_VEL
LIN {X 0,Y 105.191,Z 678.544,A -85,B 0,C 180,E1 -20824.604,E2 -20824.604} C_VEL
LIN {X 0,Y 100.426,Z 683.65,A -85,B 0,C 180,E1 -20819.332,E2 -20819.332} C_VEL
LIN {X 0,Y 96.7,Z 687.582,A -85,B 0,C 180,E1 -20813.562,E2 -20813.562} C_VEL
LIN {X 0,Y 93.903,Z 690.472,A -85,B 0,C 180,E1 -20807.42,E2 -20807.42} C_VEL
LIN {X 0,Y 92.578,Z 691.849,A -85,B 0,C 180,E1 -20803.164,E2 -20803.164} C_VEL
LIN {X 0,Y 91.678,Z 692.822,A -85,B 0,C 180,E1 -20798.819,E2 -20798.819} C_VEL
LIN {X 0,Y 91.053,Z 693.611,A -85,B 0,C 180,E1 -20790,E2 -20790} C_VEL
LIN {X 0,Y 91.678,Z 692.777,A -85,B 0,C 180,E1 -20781.181,E2 -20781.181} C_VEL
LIN {X 0,Y 92.579,Z 691.786,A -85,B 0,C 180,E1 -20776.836,E2 -20776.836} C_VEL
LIN {X 0,Y 93.909,Z 690.373,A -85,B 0,C 180,E1 -20772.581,E2 -20772.581} C_VEL
LIN {X 0,Y 96.718,Z 687.446,A -85,B 0,C 180,E1 -20766.443,E2 -20766.443} C_VEL
LIN {X 0,Y 100.474,Z 683.468,A -85,B 0,C 180,E1 -20760.683,E2 -20760.683} C_VEL
LIN {X 0,Y 105.222,Z 678.318,A -85,B 0,C 180,E1 -20755.408,E2 -20755.408} C_VEL
LIN {X 0,Y 110.682,Z 671.836,A -85,B 0,C 180,E1 -20750.582,E2 -20750.582} C_VEL
LIN {X 0,Y 116.867,Z 663.563,A -85,B 0,C 180,E1 -20746.072,E2 -20746.072} C_VEL
LIN {X 0,Y 122.22,Z 655.495,A -85,B 0,C 180,E1 -20742.848,E2 -20742.848} C_VEL
LIN {X 0,Y 128.127,Z 645.263,A -85,B 0,C 180,E1 -20739.832,E2 -20739.832} C_VEL
LIN {X 0,Y 133.674,Z 633.767,A -85,B 0,C 180,E1 -20737.325,E2 -20737.325} C_VEL
LIN {X 0,Y 138.121,Z 622.225,A -85,B 0,C 180,E1 -20735.498,E2 -20735.498} C_VEL
LIN {X 0,Y 141.739,Z 610.341,A -85,B 0,C 180,E1 -20734.164,E2 -20734.164} C_VEL
LIN {X 0,Y 144.59,Z 597.457,A -85,B 0,C 180,E1 -20733.175,E2 -20733.175} C_VEL
LIN {X 0,Y 146.424,Z 583.013,A -85,B 0,C 180,E1 -20732.501,E2 -20732.501} C_VEL
LIN {X 0,Y 147.066,Z 575.577,A -85,B 0,C 180,E1 -20732.229,E2 -20732.229} C_VEL
LIN {X 0,Y 143.369,Z 583.5,A -85,B 0,C 180,E1 -20730.57,E2 -20730.57} C_VEL
LIN {X 0,Y 139.126,Z 590.631,A -85,B 0,C 180,E1 -20728.37,E2 -20728.37} C_VEL
LIN {X 0,Y 136.536,Z 594.132,A -85,B 0,C 180,E1 -20726.872,E2 -20726.872} C_VEL
LIN {X 0,Y 131.586,Z 603.78,A -85,B 0,C 180,E1 -20724.707,E2 -20724.707} C_VEL
LIN {X 0,Y 126.253,Z 611.974,A -85,B 0,C 180,E1 -20722.109,E2 -20722.109} C_VEL
LIN {X 0,Y 121.751,Z 617.708,A -85,B 0,C 180,E1 -20719.385,E2 -20719.385} C_VEL
LIN {X 0,Y 118.876,Z 620.891,A -85,B 0,C 180,E1 -20717.194,E2 -20717.194} C_VEL
LIN {X 0,Y 117.086,Z 622.59,A -85,B 0,C 180,E1 -20715.492,E2 -20715.492} C_VEL
LIN {X 0,Y 115.686,Z 623.853,A -85,B 0,C 180,E1 -20713.909,E2 -20713.909} C_VEL
LIN {X 0,Y 111.948,Z 628.755,A -85,B 0,C 180,E1 -20710.856,E2 -20710.856} C_VEL
LIN {X 0,Y 108.785,Z 632.724,A -85,B 0,C 180,E1 -20707.424,E2 -20707.424} C_VEL
LIN {X 0,Y 107.539,Z 634.31,A -85,B 0,C 180,E1 -20705.626,E2 -20705.626} C_VEL
LIN {X 0,Y 105.356,Z 637.324,A -85,B 0,C 180,E1 -20700,E2 -20700} C_VEL
LIN {X 0,Y 102.81,Z 642.319,A -85,B 0,C 180,E1 -20694.115,E2 -20694.115} C_VEL
LIN {X 0,Y 102.251,Z 644.713,A -85,B 0,C 180,E1 -20690.106,E2 -20690.106} C_VEL
LIN {X 0,Y 103.876,Z 648.244,A -85,B 0,C 180,E1 -20681.299,E2 -20681.299} C_VEL
LIN {X 0,Y 105.343,Z 650.87,A -85,B 0,C 180,E1 -20676.404,E2 -20676.404} C_VEL
LIN {X 0,Y 107.421,Z 652.298,A -85,B 0,C 180,E1 -20672.744,E2 -20672.744} C_VEL
LIN {X 0,Y 110.442,Z 653,A -85,B 0,C 180,E1 -20669.397,E2 -20669.397} C_VEL
LIN {X 0,Y 116.827,Z 655.435,A -85,B 0,C 180,E1 -20663.018,E2 -20663.018} C_VEL
LIN {X 0,Y 122.763,Z 656.06,A -85,B 0,C 180,E1 -20659.247,E2 -20659.247} C_VEL
LIN {X 0,Y 123.731,Z 656.039,A -85,B 0,C 180,E1 -20658.766,E2 -20658.766} C_VEL
LIN {X 0,Y 123.416,Z 657.92,A -85,B 0,C 180,E1 -20657.757,E2 -20657.757} C_VEL
LIN {X 0,Y 118.126,Z 665.008,A -85,B 0,C 180,E1 -20655.557,E2 -20655.557} C_VEL
LIN {X 0,Y 112.373,Z 672.463,A -85,B 0,C 180,E1 -20652.247,E2 -20652.247} C_VEL
LIN {X 0,Y 106.948,Z 679.303,A -85,B 0,C 180,E1 -20647.948,E2 -20647.948} C_VEL
LIN {X 0,Y 102.326,Z 684.745,A -85,B 0,C 180,E1 -20643.33,E2 -20643.33} C_VEL
LIN {X 0,Y 97.97,Z 689.55,A -85,B 0,C 180,E1 -20637.794,E2 -20637.794} C_VEL
LIN {X 0,Y 94.585,Z 693.229,A -85,B 0,C 180,E1 -20631.809,E2 -20631.809} C_VEL
LIN {X 0,Y 93.006,Z 695.13,A -85,B 0,C 180,E1 -20627.593,E2 -20627.593} C_VEL
LIN {X 0,Y 91.869,Z 696.575,A -85,B 0,C 180,E1 -20623.268,E2 -20623.268} C_VEL
LIN {X 0,Y 91.191,Z 697.595,A -85,B 0,C 180,E1 -20618.867,E2 -20618.867} C_VEL
LIN {X 0,Y 90.924,Z 698.224,A -85,B 0,C 180,E1 -20614.433,E2 -20614.433} C_VEL
LIN {X 0,Y 91.045,Z 698.462,A -85,B 0,C 180,E1 -20610,E2 -20610} C_VEL
LIN {X 0,Y 91.021,Z 698.245,A -85,B 0,C 180,E1 -20605.572,E2 -20605.572} C_VEL
LIN {X 0,Y 92.253,Z 696.626,A -85,B 0,C 180,E1 -20596.788,E2 -20596.788} C_VEL
LIN {X 0,Y 93.642,Z 695.212,A -85,B 0,C 180,E1 -20592.53,E2 -20592.53} C_VEL
LIN {X 0,Y 96.692,Z 692.263,A -85,B 0,C 180,E1 -20586.436,E2 -20586.436} C_VEL
LIN {X 0,Y 100.976,Z 688.27,A -85,B 0,C 180,E1 -20580.843,E2 -20580.843} C_VEL
LIN {X 0,Y 106.538,Z 683.112,A -85,B 0,C 180,E1 -20575.894,E2 -20575.894} C_VEL
LIN {X 0,Y 108.187,Z 681.83,A -85,B 0,C 180,E1 -20574.793,E2 -20574.793} C_VEL
LIN {X 0,Y 116.027,Z 686.476,A -85,B 0,C 180,E1 -20568.218,E2 -20568.218} C_VEL
LIN {X 0,Y 120.445,Z 688.335,A -85,B 0,C 180,E1 -20565.556,E2 -20565.556} C_VEL
LIN {X 0,Y 122.202,Z 688.848,A -85,B 0,C 180,E1 -20563.641,E2 -20563.641} C_VEL
LIN {X 0,Y 113.366,Z 684.13,A -85,B 0,C 180,E1 -20558.312,E2 -20558.312} C_VEL
LIN {X 0,Y 106.302,Z 678.34,A -85,B 0,C 180,E1 -20551.932,E2 -20551.932} C_VEL
LIN {X 0,Y 101.177,Z 671.265,A -85,B 0,C 180,E1 -20544.631,E2 -20544.631} C_VEL
LIN {X 0,Y 98.559,Z 663.912,A -85,B 0,C 180,E1 -20537.641,E2 -20537.641} C_VEL
LIN {X 0,Y 97.525,Z 655.062,A -85,B 0,C 180,E1 -20530.379,E2 -20530.379} C_VEL
LIN {X 0,Y 97.305,Z 650.466,A -85,B 0,C 180,E1 -20527.131,E2 -20527.131} C_VEL
LIN {X 0,Y 96.708,Z 650.93,A -85,B 0,C 180,E1 -20526.258,E2 -20526.258} C_VEL
LIN {X 0,Y 96.341,Z 650.899,A -85,B 0,C 180,E1 -20524.183,E2 -20524.183} C_VEL
LIN {X 0,Y 96.73,Z 650.116,A -85,B 0,C 180,E1 -20522.082,E2 -20522.082} C_VEL
LIN {X 0,Y 98.415,Z 647.777,A -85,B 0,C 180,E1 -20518.778,E2 -20518.778} C_VEL
LIN {X 0,Y 98.809,Z 647.437,A -85,B 0,C 180,E1 -20515.921,E2 -20515.921} C_VEL
LIN {X 0,Y 100.931,Z 645.443,A -85,B 0,C 180,E1 -20511.995,E2 -20511.995} C_VEL
LIN {X 0,Y 103.058,Z 643.423,A -85,B 0,C 180,E1 -20509.491,E2 -20509.491} C_VEL
LIN {X 0,Y 106.529,Z 641.148,A -85,B 0,C 180,E1 -20504.699,E2 -20504.699} C_VEL
LIN {X 0,Y 108.806,Z 639.067,A -85,B 0,C 180,E1 -20503.102,E2 -20503.102} C_VEL
LIN {X 0,Y 112.224,Z 636.822,A -85,B 0,C 180,E1 -20499.947,E2 -20499.947} C_VEL
LIN {X 0,Y 115.805,Z 634.073,A -85,B 0,C 180,E1 -20497.566,E2 -20497.566} C_VEL
LIN {X 0,Y 121.158,Z 628.787,A -85,B 0,C 180,E1 -20495.13,E2 -20495.13} C_VEL
LIN {X 0,Y 125.991,Z 624.868,A -85,B 0,C 180,E1 -20492.589,E2 -20492.589} C_VEL
LIN {X 0,Y 130.148,Z 620.655,A -85,B 0,C 180,E1 -20490.922,E2 -20490.922} C_VEL
LIN {X 0,Y 134.948,Z 614.441,A -85,B 0,C 180,E1 -20489.509,E2 -20489.509} C_VEL
LIN {X 0,Y 139.669,Z 606.555,A -85,B 0,C 180,E1 -20488.408,E2 -20488.408} C_VEL
LIN {X 0,Y 141.718,Z 602.607,A -85,B 0,C 180,E1 -20487.961,E2 -20487.961} C_VEL
LIN {X 0,Y 143.277,Z 600.585,A -85,B 0,C 180,E1 -20487.353,E2 -20487.353} C_VEL
LIN {X 0,Y 143.567,Z 601.055,A -85,B 0,C 180,E1 -20487.082,E2 -20487.082} C_VEL
LIN {X 0,Y 143.214,Z 603.779,A -85,B 0,C 180,E1 -20486.76,E2 -20486.76} C_VEL
LIN {X 0,Y 140.807,Z 610.784,A -85,B 0,C 180,E1 -20486.59,E2 -20486.59} C_VEL
LIN {X 0,Y 136.063,Z 620.599,A -85,B 0,C 180,E1 -20486.672,E2 -20486.672} C_VEL
LIN {X 0,Y 132.472,Z 627.775,A -85,B 0,C 180,E1 -20486.287,E2 -20486.287} C_VEL
LIN {X 0,Y 131.404,Z 630.128,A -85,B 0,C 180,E1 -20485.964,E2 -20485.964} C_VEL
LIN {X 0,Y 126.211,Z 641.227,A -85,B 0,C 180,E1 -20483.845,E2 -20483.845} C_VEL
LIN {X 0,Y 120.498,Z 651.324,A -85,B 0,C 180,E1 -20481.269,E2 -20481.269} C_VEL
LIN {X 0,Y 115.053,Z 659.582,A -85,B 0,C 180,E1 -20478.443,E2 -20478.443} C_VEL
LIN {X 0,Y 108.396,Z 668.506,A -85,B 0,C 180,E1 -20474.186,E2 -20474.186} C_VEL
LIN {X 0,Y 102.289,Z 675.688,A -85,B 0,C 180,E1 -20469.46,E2 -20469.46} C_VEL
LIN {X 0,Y 97.628,Z 680.549,A -85,B 0,C 180,E1 -20465.163,E2 -20465.163} C_VEL
LIN {X 0,Y 92.846,Z 685.246,A -85,B 0,C 180,E1 -20459.473,E2 -20459.473} C_VEL
LIN {X 0,Y 89.096,Z 688.821,A -85,B 0,C 180,E1 -20453.229,E2 -20453.229} C_VEL
LIN {X 0,Y 87.161,Z 690.66,A -85,B 0,C 180,E1 -20448.816,E2 -20448.816} C_VEL
LIN {X 0,Y 85.668,Z 692.038,A -85,B 0,C 180,E1 -20444.248,E2 -20444.248} C_VEL
LIN {X 0,Y 84.669,Z 693.01,A -85,B 0,C 180,E1 -20439.556,E2 -20439.556} C_VEL
LIN {X 0,Y 84.072,Z 693.602,A -85,B 0,C 180,E1 -20434.795,E2 -20434.795} C_VEL
LIN {X 0,Y 83.954,Z 693.801,A -85,B 0,C 180,E1 -20430,E2 -20430} C_VEL
LIN {X 0,Y 84.669,Z 692.966,A -85,B 0,C 180,E1 -20420.444,E2 -20420.444} C_VEL
LIN {X 0,Y 85.669,Z 691.976,A -85,B 0,C 180,E1 -20415.753,E2 -20415.753} C_VEL
LIN {X 0,Y 87.167,Z 690.563,A -85,B 0,C 180,E1 -20411.185,E2 -20411.185} C_VEL
LIN {X 0,Y 90.253,Z 687.635,A -85,B 0,C 180,E1 -20404.641,E2 -20404.641} C_VEL
LIN {X 0,Y 94.334,Z 683.657,A -85,B 0,C 180,E1 -20398.566,E2 -20398.566} C_VEL
LIN {X 0,Y 99.457,Z 678.506,A -85,B 0,C 180,E1 -20393.084,E2 -20393.084} C_VEL
LIN {X 0,Y 105.29,Z 672.024,A -85,B 0,C 180,E1 -20388.126,E2 -20388.126} C_VEL
LIN {X 0,Y 111.693,Z 663.964,A -85,B 0,C 180,E1 -20383.649,E2 -20383.649} C_VEL
LIN {X 0,Y 117.514,Z 655.68,A -85,B 0,C 180,E1 -20380.313,E2 -20380.313} C_VEL
LIN {X 0,Y 123.706,Z 645.446,A -85,B 0,C 180,E1 -20377.31,E2 -20377.31} C_VEL
LIN {X 0,Y 129.497,Z 633.947,A -85,B 0,C 180,E1 -20374.829,E2 -20374.829} C_VEL
LIN {X 0,Y 134.131,Z 622.399,A -85,B 0,C 180,E1 -20373.034,E2 -20373.034} C_VEL
LIN {X 0,Y 137.972,Z 610.158,A -85,B 0,C 180,E1 -20371.688,E2 -20371.688} C_VEL
LIN {X 0,Y 140.801,Z 597.813,A -85,B 0,C 180,E1 -20370.774,E2 -20370.774} C_VEL
LIN {X 0,Y 141.219,Z 594.916,A -85,B 0,C 180,E1 -20370.574,E2 -20370.574} C_VEL
LIN {X 0,Y 138.042,Z 599.012,A -85,B 0,C 180,E1 -20369.028,E2 -20369.028} C_VEL
LIN {X 0,Y 132.192,Z 608.973,A -85,B 0,C 180,E1 -20366.866,E2 -20366.866} C_VEL
LIN {X 0,Y 126.71,Z 616.478,A -85,B 0,C 180,E1 -20364.582,E2 -20364.582} C_VEL
LIN {X 0,Y 120.877,Z 623.108,A -85,B 0,C 180,E1 -20361.523,E2 -20361.523} C_VEL
LIN {X 0,Y 117.451,Z 626.433,A -85,B 0,C 180,E1 -20359.215,E2 -20359.215} C_VEL
LIN {X 0,Y 113.684,Z 629.678,A -85,B 0,C 180,E1 -20355.881,E2 -20355.881} C_VEL
LIN {X 0,Y 108.768,Z 635.173,A -85,B 0,C 180,E1 -20352.122,E2 -20352.122} C_VEL
LIN {X 0,Y 104.696,Z 639.516,A -85,B 0,C 180,E1 -20347.716,E2 -20347.716} C_VEL
LIN {X 0,Y 101.771,Z 642.751,A -85,B 0,C 180,E1 -20341.652,E2 -20341.652} C_VEL
LIN {X 0,Y 98.702,Z 647.586,A -85,B 0,C 180,E1 -20335.458,E2 -20335.458} C_VEL
LIN {X 0,Y 97.945,Z 649.654,A -85,B 0,C 180,E1 -20331.749,E2 -20331.749} C_VEL
LIN {X 0,Y 98.699,Z 652.807,A -85,B 0,C 180,E1 -20323.452,E2 -20323.452} C_VEL
LIN {X 0,Y 101.753,Z 656.924,A -85,B 0,C 180,E1 -20313.884,E2 -20313.884} C_VEL
LIN {X 0,Y 109.491,Z 659.565,A -85,B 0,C 180,E1 -20304.712,E2 -20304.712} C_VEL
LIN {X 0,Y 112.988,Z 660.654,A -85,B 0,C 180,E1 -20301.537,E2 -20301.537} C_VEL
LIN {X 0,Y 115.361,Z 660.969,A -85,B 0,C 180,E1 -20299.915,E2 -20299.915} C_VEL
LIN {X 0,Y 115.463,Z 662.037,A -85,B 0,C 180,E1 -20299.067,E2 -20299.067} C_VEL
LIN {X 0,Y 109.555,Z 669.456,A -85,B 0,C 180,E1 -20296.194,E2 -20296.194} C_VEL
LIN {X 0,Y 102.912,Z 677.352,A -85,B 0,C 180,E1 -20291.746,E2 -20291.746} C_VEL
LIN {X 0,Y 98.234,Z 682.693,A -85,B 0,C 180,E1 -20287.454,E2 -20287.454} C_VEL
LIN {X 0,Y 93.17,Z 687.909,A -85,B 0,C 180,E1 -20281.872,E2 -20281.872} C_VEL
LIN {X 0,Y 89.119,Z 691.952,A -85,B 0,C 180,E1 -20275.705,E2 -20275.705} C_VEL
LIN {X 0,Y 86.237,Z 694.939,A -85,B 0,C 180,E1 -20269.025,E2 -20269.025} C_VEL
LIN {X 0,Y 84.956,Z 696.385,A -85,B 0,C 180,E1 -20264.37,E2 -20264.37} C_VEL
LIN {X 0,Y 84.167,Z 697.405,A -85,B 0,C 180,E1 -20259.614,E2 -20259.614} C_VEL
LIN {X 0,Y 83.828,Z 698.035,A -85,B 0,C 180,E1 -20254.809,E2 -20254.809} C_VEL
LIN {X 0,Y 83.944,Z 698.273,A -85,B 0,C 180,E1 -20250,E2 -20250} C_VEL
LIN {X 0,Y 83.935,Z 698.056,A -85,B 0,C 180,E1 -20245.197,E2 -20245.197} C_VEL
LIN {X 0,Y 85.346,Z 696.437,A -85,B 0,C 180,E1 -20235.698,E2 -20235.698} C_VEL
LIN {X 0,Y 86.882,Z 695.023,A -85,B 0,C 180,E1 -20231.121,E2 -20231.121} C_VEL
LIN {X 0,Y 90.23,Z 692.075,A -85,B 0,C 180,E1 -20224.634,E2 -20224.634} C_VEL
LIN {X 0,Y 94.837,Z 688.083,A -85,B 0,C 180,E1 -20218.752,E2 -20218.752} C_VEL
LIN {X 0,Y 100.743,Z 682.927,A -85,B 0,C 180,E1 -20213.631,E2 -20213.631} C_VEL
LIN {X 0,Y 104.291,Z 679.913,A -85,B 0,C 180,E1 -20211.439,E2 -20211.439} C_VEL
LIN {X 0,Y 112.607,Z 684.702,A -85,B 0,C 180,E1 -20205.03,E2 -20205.03} C_VEL
LIN {X 0,Y 113.718,Z 685.17,A -85,B 0,C 180,E1 -20204.005,E2 -20204.005} C_VEL
LIN {X 0,Y 106.152,Z 680.405,A -85,B 0,C 180,E1 -20198.974,E2 -20198.974} C_VEL
LIN {X 0,Y 97.836,Z 672.051,A -85,B 0,C 180,E1 -20190.188,E2 -20190.188} C_VEL
LIN {X 0,Y 93.636,Z 663.818,A -85,B 0,C 180,E1 -20182.042,E2 -20182.042} C_VEL
LIN {X 0,Y 92.606,Z 660.891,A -85,B 0,C 180,E1 -20179.104,E2 -20179.104} C_VEL
LIN {X 0,Y 91.72,Z 661.034,A -85,B 0,C 180,E1 -20177.848,E2 -20177.848} C_VEL
LIN {X 0,Y 90.699,Z 659.949,A -85,B 0,C 180,E1 -20173.442,E2 -20173.442} C_VEL
LIN {X 0,Y 91.387,Z 657.648,A -85,B 0,C 180,E1 -20168.847,E2 -20168.847} C_VEL
LIN {X 0,Y 92.049,Z 656.413,A -85,B 0,C 180,E1 -20166.991,E2 -20166.991} C_VEL
LIN {X 0,Y 91.69,Z 656.246,A -85,B 0,C 180,E1 -20164.396,E2 -20164.396} C_VEL
LIN {X 0,Y 92.596,Z 654.785,A -85,B 0,C 180,E1 -20160,E2 -20160} C_VEL
LIN {X 0,Y 97.703,Z 650.253,A -85,B 0,C 180,E1 -20149.64,E2 -20149.64} C_VEL
LIN {X 0,Y 99.509,Z 648.792,A -85,B 0,C 180,E1 -20147.767,E2 -20147.767} C_VEL
LIN {X 0,Y 104.039,Z 646.097,A -85,B 0,C 180,E1 -20142.303,E2 -20142.303} C_VEL
LIN {X 0,Y 106.484,Z 644.169,A -85,B 0,C 180,E1 -20140.731,E2 -20140.731} C_VEL
LIN {X 0,Y 110.39,Z 641.859,A -85,B 0,C 180,E1 -20137.543,E2 -20137.543} C_VEL
LIN {X 0,Y 112.711,Z 640.308,A -85,B 0,C 180,E1 -20136.09,E2 -20136.09} C_VEL
LIN {X 0,Y 115.316,Z 638.344,A -85,B 0,C 180,E1 -20134.747,E2 -20134.747} C_VEL
LIN {X 0,Y 121.147,Z 633.315,A -85,B 0,C 180,E1 -20132.348,E2 -20132.348} C_VEL
LIN {X 0,Y 126.51,Z 629.188,A -85,B 0,C 180,E1 -20130.001,E2 -20130.001} C_VEL
LIN {X 0,Y 131.2,Z 624.755,A -85,B 0,C 180,E1 -20128.424,E2 -20128.424} C_VEL
LIN {X 0,Y 134.587,Z 620.822,A -85,B 0,C 180,E1 -20127.552,E2 -20127.552} C_VEL
LIN {X 0,Y 134.533,Z 622.036,A -85,B 0,C 180,E1 -20127.143,E2 -20127.143} C_VEL
LIN {X 0,Y 131.404,Z 630.128,A -85,B 0,C 180,E1 -20125.964,E2 -20125.964} C_VEL
LIN {X 0,Y 128.74,Z 635.301,A -85,B 0,C 180,E1 -20125.314,E2 -20125.314} C_VEL
LIN {X 0,Y 123.041,Z 643.355,A -85,B 0,C 180,E1 -20124.737,E2 -20124.737} C_VEL
LIN {X 0,Y 116.923,Z 650.902,A -85,B 0,C 180,E1 -20123.915,E2 -20123.915} C_VEL
LIN {X 0,Y 113.651,Z 655.244,A -85,B 0,C 180,E1 -20122.84,E2 -20122.84} C_VEL
LIN {X 0,Y 108.067,Z 662.964,A -85,B 0,C 180,E1 -20119.83,E2 -20119.83} C_VEL
LIN {X 0,Y 101.057,Z 671.376,A -85,B 0,C 180,E1 -20115.34,E2 -20115.34} C_VEL
LIN {X 0,Y 95.869,Z 676.933,A -85,B 0,C 180,E1 -20111.283,E2 -20111.283} C_VEL
LIN {X 0,Y 90.047,Z 682.441,A -85,B 0,C 180,E1 -20105.829,E2 -20105.829} C_VEL
LIN {X 0,Y 85.261,Z 686.745,A -85,B 0,C 180,E1 -20099.642,E2 -20099.642} C_VEL
LIN {X 0,Y 82.613,Z 689.009,A -85,B 0,C 180,E1 -20095.173,E2 -20095.173} C_VEL
LIN {X 0,Y 80.456,Z 690.849,A -85,B 0,C 180,E1 -20090.451,E2 -20090.451} C_VEL
LIN {X 0,Y 78.808,Z 692.226,A -85,B 0,C 180,E1 -20085.518,E2 -20085.518} C_VEL
LIN {X 0,Y 77.691,Z 693.199,A -85,B 0,C 180,E1 -20080.424,E2 -20080.424} C_VEL
LIN {X 0,Y 77.008,Z 693.79,A -85,B 0,C 180,E1 -20075.236,E2 -20075.236} C_VEL
LIN {X 0,Y 76.882,Z 693.989,A -85,B 0,C 180,E1 -20070,E2 -20070} C_VEL
LIN {X 0,Y 77.691,Z 693.155,A -85,B 0,C 180,E1 -20059.577,E2 -20059.577} C_VEL
LIN {X 0,Y 78.809,Z 692.165,A -85,B 0,C 180,E1 -20054.482,E2 -20054.482} C_VEL
LIN {X 0,Y 80.461,Z 690.753,A -85,B 0,C 180,E1 -20049.55,E2 -20049.55} C_VEL
LIN {X 0,Y 83.878,Z 687.825,A -85,B 0,C 180,E1 -20042.559,E2 -20042.559} C_VEL
LIN {X 0,Y 88.341,Z 683.847,A -85,B 0,C 180,E1 -20036.159,E2 -20036.159} C_VEL
LIN {X 0,Y 93.868,Z 678.695,A -85,B 0,C 180,E1 -20030.475,E2 -20030.475} C_VEL
LIN {X 0,Y 100.107,Z 672.213,A -85,B 0,C 180,E1 -20025.408,E2 -20025.408} C_VEL
LIN {X 0,Y 106.918,Z 664.151,A -85,B 0,C 180,E1 -20020.896,E2 -20020.896} C_VEL
LIN {X 0,Y 113.045,Z 655.866,A -85,B 0,C 180,E1 -20017.564,E2 -20017.564} C_VEL
LIN {X 0,Y 119.544,Z 645.629,A -85,B 0,C 180,E1 -20014.607,E2 -20014.607} C_VEL
LIN {X 0,Y 125.591,Z 634.126,A -85,B 0,C 180,E1 -20012.179,E2 -20012.179} C_VEL
LIN {X 0,Y 130.398,Z 622.575,A -85,B 0,C 180,E1 -20010.418,E2 -20010.418} C_VEL
LIN {X 0,Y 132.991,Z 615.119,A -85,B 0,C 180,E1 -20009.588,E2 -20009.588} C_VEL
LIN {X 0,Y 133.239,Z 613.452,A -85,B 0,C 180,E1 -20009.204,E2 -20009.204} C_VEL
LIN {X 0,Y 127.305,Z 620.833,A -85,B 0,C 180,E1 -20007.094,E2 -20007.094} C_VEL
LIN {X 0,Y 120.582,Z 627.77,A -85,B 0,C 180,E1 -20004.079,E2 -20004.079} C_VEL
LIN {X 0,Y 115.916,Z 631.838,A -85,B 0,C 180,E1 -20001.333,E2 -20001.333} C_VEL
LIN {X 0,Y 112.03,Z 634.805,A -85,B 0,C 180,E1 -19998.281,E2 -19998.281} C_VEL
LIN {X 0,Y 107.363,Z 639.362,A -85,B 0,C 180,E1 -19995.18,E2 -19995.18} C_VEL
LIN {X 0,Y 103.376,Z 643.04,A -85,B 0,C 180,E1 -19991.769,E2 -19991.769} C_VEL
LIN {X 0,Y 100.353,Z 645.75,A -85,B 0,C 180,E1 -19988.052,E2 -19988.052} C_VEL
LIN {X 0,Y 98.294,Z 647.661,A -85,B 0,C 180,E1 -19984.1,E2 -19984.1} C_VEL
LIN {X 0,Y 97.161,Z 648.988,A -85,B 0,C 180,E1 -19982.073,E2 -19982.073} C_VEL
LIN {X 0,Y 94.774,Z 652.05,A -85,B 0,C 180,E1 -19977.875,E2 -19977.875} C_VEL
LIN {X 0,Y 93.986,Z 653.32,A -85,B 0,C 180,E1 -19975.712,E2 -19975.712} C_VEL
LIN {X 0,Y 93.136,Z 656.227,A -85,B 0,C 180,E1 -19968.806,E2 -19968.806} C_VEL
LIN {X 0,Y 93.939,Z 658.375,A -85,B 0,C 180,E1 -19962.587,E2 -19962.587} C_VEL
LIN {X 0,Y 96.42,Z 661.679,A -85,B 0,C 180,E1 -19954.066,E2 -19954.066} C_VEL
LIN {X 0,Y 106.671,Z 665.013,A -85,B 0,C 180,E1 -19941.818,E2 -19941.818} C_VEL
LIN {X 0,Y 107.646,Z 665.867,A -85,B 0,C 180,E1 -19940.44,E2 -19940.44} C_VEL
LIN {X 0,Y 101.106,Z 673.429,A -85,B 0,C 180,E1 -19936.876,E2 -19936.876} C_VEL
LIN {X 0,Y 94.618,Z 680.495,A -85,B 0,C 180,E1 -19931.951,E2 -19931.951} C_VEL
LIN {X 0,Y 88.913,Z 686.112,A -85,B 0,C 180,E1 -19926.358,E2 -19926.358} C_VEL
LIN {X 0,Y 84.124,Z 690.523,A -85,B 0,C 180,E1 -19920.083,E2 -19920.083} C_VEL
LIN {X 0,Y 81.499,Z 692.848,A -85,B 0,C 180,E1 -19915.542,E2 -19915.542} C_VEL
LIN {X 0,Y 79.519,Z 694.749,A -85,B 0,C 180,E1 -19910.703,E2 -19910.703} C_VEL
LIN {X 0,Y 78.06,Z 696.195,A -85,B 0,C 180,E1 -19905.67,E2 -19905.67} C_VEL
LIN {X 0,Y 77.148,Z 697.215,A -85,B 0,C 180,E1 -19900.498,E2 -19900.498} C_VEL
LIN {X 0,Y 76.756,Z 697.845,A -85,B 0,C 180,E1 -19895.254,E2 -19895.254} C_VEL
LIN {X 0,Y 76.849,Z 698.084,A -85,B 0,C 180,E1 -19890,E2 -19890} C_VEL
LIN {X 0,Y 76.873,Z 697.867,A -85,B 0,C 180,E1 -19884.754,E2 -19884.754} C_VEL
LIN {X 0,Y 78.486,Z 696.249,A -85,B 0,C 180,E1 -19874.417,E2 -19874.417} C_VEL
LIN {X 0,Y 80.192,Z 694.835,A -85,B 0,C 180,E1 -19869.478,E2 -19869.478} C_VEL
LIN {X 0,Y 83.875,Z 691.888,A -85,B 0,C 180,E1 -19862.558,E2 -19862.558} C_VEL
LIN {X 0,Y 88.843,Z 687.896,A -85,B 0,C 180,E1 -19856.376,E2 -19856.376} C_VEL
LIN {X 0,Y 95.128,Z 682.742,A -85,B 0,C 180,E1 -19851.099,E2 -19851.099} C_VEL
LIN {X 0,Y 100.888,Z 677.983,A -85,B 0,C 180,E1 -19847.726,E2 -19847.726} C_VEL
LIN {X 0,Y 103.862,Z 679.823,A -85,B 0,C 180,E1 -19845.373,E2 -19845.373} C_VEL
LIN {X 0,Y 104.382,Z 680.007,A -85,B 0,C 180,E1 -19843.688,E2 -19843.688} C_VEL
LIN {X 0,Y 97.283,Z 674.382,A -85,B 0,C 180,E1 -19837.884,E2 -19837.884} C_VEL
LIN {X 0,Y 93.174,Z 670.028,A -85,B 0,C 180,E1 -19833.285,E2 -19833.285} C_VEL
LIN {X 0,Y 92.001,Z 670.099,A -85,B 0,C 180,E1 -19832.326,E2 -19832.326} C_VEL
LIN {X 0,Y 89.069,Z 669.326,A -85,B 0,C 180,E1 -19828.257,E2 -19828.257} C_VEL
LIN {X 0,Y 86.807,Z 665.877,A -85,B 0,C 180,E1 -19818.895,E2 -19818.895} C_VEL
LIN {X 0,Y 85.604,Z 664.933,A -85,B 0,C 180,E1 -19814.258,E2 -19814.258} C_VEL
LIN {X 0,Y 86.769,Z 661.318,A -85,B 0,C 180,E1 -19804.646,E2 -19804.646} C_VEL
LIN {X 0,Y 87.543,Z 660.083,A -85,B 0,C 180,E1 -19800,E2 -19800} C_VEL
LIN {X 0,Y 93.247,Z 655.66,A -85,B 0,C 180,E1 -19788.466,E2 -19788.466} C_VEL
LIN {X 0,Y 96.289,Z 653.622,A -85,B 0,C 180,E1 -19785.199,E2 -19785.199} C_VEL
LIN {X 0,Y 101.499,Z 650.874,A -85,B 0,C 180,E1 -19779.744,E2 -19779.744} C_VEL
LIN {X 0,Y 104.106,Z 649.065,A -85,B 0,C 180,E1 -19778.204,E2 -19778.204} C_VEL
LIN {X 0,Y 108.574,Z 646.69,A -85,B 0,C 180,E1 -19774.989,E2 -19774.989} C_VEL
LIN {X 0,Y 112.975,Z 643.901,A -85,B 0,C 180,E1 -19772.721,E2 -19772.721} C_VEL
LIN {X 0,Y 119.916,Z 638.59,A -85,B 0,C 180,E1 -19770.121,E2 -19770.121} C_VEL
LIN {X 0,Y 123.399,Z 636.201,A -85,B 0,C 180,E1 -19768.683,E2 -19768.683} C_VEL
LIN {X 0,Y 124.87,Z 636.134,A -85,B 0,C 180,E1 -19767.591,E2 -19767.591} C_VEL
LIN {X 0,Y 118.811,Z 647.292,A -85,B 0,C 180,E1 -19765.16,E2 -19765.16} C_VEL
LIN {X 0,Y 113.651,Z 655.244,A -85,B 0,C 180,E1 -19762.84,E2 -19762.84} C_VEL
LIN {X 0,Y 110.269,Z 659.47,A -85,B 0,C 180,E1 -19761.609,E2 -19761.609} C_VEL
LIN {X 0,Y 103.413,Z 665.977,A -85,B 0,C 180,E1 -19759.968,E2 -19759.968} C_VEL
LIN {X 0,Y 96.342,Z 671.869,A -85,B 0,C 180,E1 -19757.858,E2 -19757.858} C_VEL
LIN {X 0,Y 92.722,Z 675.121,A -85,B 0,C 180,E1 -19755.833,E2 -19755.833} C_VEL
LIN {X 0,Y 86.392,Z 680.922,A -85,B 0,C 180,E1 -19750.602,E2 -19750.602} C_VEL
LIN {X 0,Y 80.757,Z 685.621,A -85,B 0,C 180,E1 -19744.449,E2 -19744.449} C_VEL
LIN {X 0,Y 76.226,Z 689.197,A -85,B 0,C 180,E1 -19737.452,E2 -19737.452} C_VEL
LIN {X 0,Y 73.838,Z 691.037,A -85,B 0,C 180,E1 -19732.379,E2 -19732.379} C_VEL
LIN {X 0,Y 72.002,Z 692.415,A -85,B 0,C 180,E1 -19727.027,E2 -19727.027} C_VEL
LIN {X 0,Y 70.709,Z 693.388,A -85,B 0,C 180,E1 -19721.466,E2 -19721.466} C_VEL
LIN {X 0,Y 69.94,Z 693.979,A -85,B 0,C 180,E1 -19715.767,E2 -19715.767} C_VEL
LIN {X 0,Y 69.783,Z 694.178,A -85,B 0,C 180,E1 -19710,E2 -19710} C_VEL
LIN {X 0,Y 70.71,Z 693.344,A -85,B 0,C 180,E1 -19698.534,E2 -19698.534} C_VEL
LIN {X 0,Y 72.004,Z 692.354,A -85,B 0,C 180,E1 -19692.973,E2 -19692.973} C_VEL
LIN {X 0,Y 73.843,Z 690.942,A -85,B 0,C 180,E1 -19687.623,E2 -19687.623} C_VEL
LIN {X 0,Y 77.639,Z 688.015,A -85,B 0,C 180,E1 -19680.141,E2 -19680.141} C_VEL
LIN {X 0,Y 82.526,Z 684.036,A -85,B 0,C 180,E1 -19673.407,E2 -19673.407} C_VEL
LIN {X 0,Y 88.504,Z 678.884,A -85,B 0,C 180,E1 -19667.548,E2 -19667.548} C_VEL
LIN {X 0,Y 95.172,Z 672.401,A -85,B 0,C 180,E1 -19662.4,E2 -19662.4} C_VEL
LIN {X 0,Y 102.159,Z 664.627,A -85,B 0,C 180,E1 -19658.029,E2 -19658.029} C_VEL
LIN {X 0,Y 108.855,Z 656.052,A -85,B 0,C 180,E1 -19654.596,E2 -19654.596} C_VEL
LIN {X 0,Y 115.667,Z 645.813,A -85,B 0,C 180,E1 -19651.717,E2 -19651.717} C_VEL
LIN {X 0,Y 121.961,Z 634.308,A -85,B 0,C 180,E1 -19649.358,E2 -19649.358} C_VEL
LIN {X 0,Y 124.3,Z 629.327,A -85,B 0,C 180,E1 -19648.582,E2 -19648.582} C_VEL
LIN {X 0,Y 124.534,Z 628.501,A -85,B 0,C 180,E1 -19648.36,E2 -19648.36} C_VEL
LIN {X 0,Y 118.026,Z 634.263,A -85,B 0,C 180,E1 -19645.576,E2 -19645.576} C_VEL
LIN {X 0,Y 114.53,Z 636.92,A -85,B 0,C 180,E1 -19643.699,E2 -19643.699} C_VEL
LIN {X 0,Y 109.978,Z 640.063,A -85,B 0,C 180,E1 -19640.578,E2 -19640.578} C_VEL
LIN {X 0,Y 102.616,Z 646.268,A -85,B 0,C 180,E1 -19635.9,E2 -19635.9} C_VEL
LIN {X 0,Y 98.667,Z 649.406,A -85,B 0,C 180,E1 -19632.339,E2 -19632.339} C_VEL
LIN {X 0,Y 93.34,Z 653.703,A -85,B 0,C 180,E1 -19624.318,E2 -19624.318} C_VEL
LIN {X 0,Y 90.578,Z 656.614,A -85,B 0,C 180,E1 -19620,E2 -19620} C_VEL
LIN {X 0,Y 88.901,Z 658.847,A -85,B 0,C 180,E1 -19615.466,E2 -19615.466} C_VEL
LIN {X 0,Y 88.146,Z 660.634,A -85,B 0,C 180,E1 -19610.824,E2 -19610.824} C_VEL
LIN {X 0,Y 91.683,Z 666.606,A -85,B 0,C 180,E1 -19592.617,E2 -19592.617} C_VEL
LIN {X 0,Y 99.693,Z 669.02,A -85,B 0,C 180,E1 -19582.517,E2 -19582.517} C_VEL
LIN {X 0,Y 98.953,Z 670.548,A -85,B 0,C 180,E1 -19581.376,E2 -19581.376} C_VEL
LIN {X 0,Y 91.627,Z 678.103,A -85,B 0,C 180,E1 -19576.776,E2 -19576.776} C_VEL
LIN {X 0,Y 85.3,Z 684.178,A -85,B 0,C 180,E1 -19571.234,E2 -19571.234} C_VEL
LIN {X 0,Y 79.68,Z 688.98,A -85,B 0,C 180,E1 -19564.982,E2 -19564.982} C_VEL
LIN {X 0,Y 75.126,Z 692.658,A -85,B 0,C 180,E1 -19557.888,E2 -19557.888} C_VEL
LIN {X 0,Y 72.89,Z 694.558,A -85,B 0,C 180,E1 -19552.686,E2 -19552.686} C_VEL
LIN {X 0,Y 71.222,Z 696.005,A -85,B 0,C 180,E1 -19547.219,E2 -19547.219} C_VEL
LIN {X 0,Y 70.163,Z 697.025,A -85,B 0,C 180,E1 -19541.556,E2 -19541.556} C_VEL
LIN {X 0,Y 69.668,Z 697.656,A -85,B 0,C 180,E1 -19535.79,E2 -19535.79} C_VEL
LIN {X 0,Y 69.747,Z 697.895,A -85,B 0,C 180,E1 -19530,E2 -19530} C_VEL
LIN {X 0,Y 69.802,Z 697.678,A -85,B 0,C 180,E1 -19524.221,E2 -19524.221} C_VEL
LIN {X 0,Y 71.681,Z 696.061,A -85,B 0,C 180,E1 -19512.894,E2 -19512.894} C_VEL
LIN {X 0,Y 73.586,Z 694.647,A -85,B 0,C 180,E1 -19507.541,E2 -19507.541} C_VEL
LIN {X 0,Y 77.654,Z 691.701,A -85,B 0,C 180,E1 -19500.147,E2 -19500.147} C_VEL
LIN {X 0,Y 83.024,Z 687.71,A -85,B 0,C 180,E1 -19493.661,E2 -19493.661} C_VEL
LIN {X 0,Y 89.724,Z 682.556,A -85,B 0,C 180,E1 -19488.257,E2 -19488.257} C_VEL
LIN {X 0,Y 95.731,Z 677.697,A -85,B 0,C 180,E1 -19484.838,E2 -19484.838} C_VEL
LIN {X 0,Y 95.007,Z 676.907,A -85,B 0,C 180,E1 -19483.427,E2 -19483.427} C_VEL
LIN {X 0,Y 90.171,Z 675.635,A -85,B 0,C 180,E1 -19478.574,E2 -19478.574} C_VEL
LIN {X 0,Y 87.258,Z 674.364,A -85,B 0,C 180,E1 -19474.319,E2 -19474.319} C_VEL
LIN {X 0,Y 84.115,Z 673.687,A -85,B 0,C 180,E1 -19470.087,E2 -19470.087} C_VEL
LIN {X 0,Y 82.195,Z 672.368,A -85,B 0,C 180,E1 -19465.31,E2 -19465.31} C_VEL
LIN {X 0,Y 81.28,Z 670.698,A -85,B 0,C 180,E1 -19460.235,E2 -19460.235} C_VEL
LIN {X 0,Y 80.207,Z 668.177,A -85,B 0,C 180,E1 -19450.093,E2 -19450.093} C_VEL
LIN {X 0,Y 81.185,Z 666.402,A -85,B 0,C 180,E1 -19444.966,E2 -19444.966} C_VEL
LIN {X 0,Y 86.266,Z 662.078,A -85,B 0,C 180,E1 -19430.622,E2 -19430.622} C_VEL
LIN {X 0,Y 91.081,Z 659.305,A -85,B 0,C 180,E1 -19424.331,E2 -19424.331} C_VEL
LIN {X 0,Y 99.451,Z 655.139,A -85,B 0,C 180,E1 -19416.735,E2 -19416.735} C_VEL
LIN {X 0,Y 101.702,Z 653.774,A -85,B 0,C 180,E1 -19415.504,E2 -19415.504} C_VEL
LIN {X 0,Y 106.438,Z 651.52,A -85,B 0,C 180,E1 -19412.47,E2 -19412.47} C_VEL
LIN {X 0,Y 109.111,Z 650.061,A -85,B 0,C 180,E1 -19411.113,E2 -19411.113} C_VEL
LIN {X 0,Y 114.937,Z 646.354,A -85,B 0,C 180,E1 -19408.877,E2 -19408.877} C_VEL
LIN {X 0,Y 115.603,Z 646.323,A -85,B 0,C 180,E1 -19408.334,E2 -19408.334} C_VEL
LIN {X 0,Y 108.78,Z 656.458,A -85,B 0,C 180,E1 -19405.462,E2 -19405.462} C_VEL
LIN {X 0,Y 101.118,Z 666.112,A -85,B 0,C 180,E1 -19401.436,E2 -19401.436} C_VEL
LIN {X 0,Y 94,Z 673.86,A -85,B 0,C 180,E1 -19396.8,E2 -19396.8} C_VEL
LIN {X 0,Y 92.722,Z 675.121,A -85,B 0,C 180,E1 -19395.833,E2 -19395.833} C_VEL
LIN {X 0,Y 89.104,Z 678.169,A -85,B 0,C 180,E1 -19393.599,E2 -19393.599} C_VEL
LIN {X 0,Y 81.858,Z 682.714,A -85,B 0,C 180,E1 -19390.233,E2 -19390.233} C_VEL
LIN {X 0,Y 74.702,Z 686.534,A -85,B 0,C 180,E1 -19386.048,E2 -19386.048} C_VEL
LIN {X 0,Y 71.412,Z 688.419,A -85,B 0,C 180,E1 -19382.496,E2 -19382.496} C_VEL
LIN {X 0,Y 67.327,Z 691.225,A -85,B 0,C 180,E1 -19374.68,E2 -19374.68} C_VEL
LIN {X 0,Y 65.239,Z 692.603,A -85,B 0,C 180,E1 -19368.855,E2 -19368.855} C_VEL
LIN {X 0,Y 63.761,Z 693.577,A -85,B 0,C 180,E1 -19362.735,E2 -19362.735} C_VEL
LIN {X 0,Y 62.898,Z 694.168,A -85,B 0,C 180,E1 -19356.415,E2 -19356.415} C_VEL
LIN {X 0,Y 62.699,Z 694.367,A -85,B 0,C 180,E1 -19350,E2 -19350} C_VEL
LIN {X 0,Y 63.761,Z 693.534,A -85,B 0,C 180,E1 -19337.265,E2 -19337.265} C_VEL
LIN {X 0,Y 65.241,Z 692.544,A -85,B 0,C 180,E1 -19331.145,E2 -19331.145} C_VEL
LIN {X 0,Y 67.332,Z 691.132,A -85,B 0,C 180,E1 -19325.322,E2 -19325.322} C_VEL
LIN {X 0,Y 71.565,Z 688.204,A -85,B 0,C 180,E1 -19317.308,E2 -19317.308} C_VEL
LIN {X 0,Y 76.935,Z 684.226,A -85,B 0,C 180,E1 -19310.249,E2 -19310.249} C_VEL
LIN {X 0,Y 83.404,Z 679.073,A -85,B 0,C 180,E1 -19304.254,E2 -19304.254} C_VEL
LIN {X 0,Y 90.532,Z 672.59,A -85,B 0,C 180,E1 -19299.077,E2 -19299.077} C_VEL
LIN {X 0,Y 98.203,Z 664.522,A -85,B 0,C 180,E1 -19294.612,E2 -19294.612} C_VEL
LIN {X 0,Y 104.988,Z 656.237,A -85,B 0,C 180,E1 -19291.405,E2 -19291.405} C_VEL
LIN {X 0,Y 112.105,Z 645.996,A -85,B 0,C 180,E1 -19288.636,E2 -19288.636} C_VEL
LIN {X 0,Y 114.519,Z 641.998,A -85,B 0,C 180,E1 -19287.746,E2 -19287.746} C_VEL
LIN {X 0,Y 115.191,Z 640.433,A -85,B 0,C 180,E1 -19287.199,E2 -19287.199} C_VEL
LIN {X 0,Y 107.863,Z 645.135,A -85,B 0,C 180,E1 -19283.013,E2 -19283.013} C_VEL
LIN {X 0,Y 99.935,Z 651.029,A -85,B 0,C 180,E1 -19278.45,E2 -19278.45} C_VEL
LIN {X 0,Y 95.353,Z 654.191,A -85,B 0,C 180,E1 -19274.731,E2 -19274.731} C_VEL
LIN {X 0,Y 89.424,Z 658.21,A -85,B 0,C 180,E1 -19266.77,E2 -19266.77} C_VEL
